LIN {X 0,Y 433.685,Z 905.49,A -85,B 0,C 180,E1 20760.988,E2 20760.988} C_VEL
LIN {X 0,Y 436.129,Z 886.958,A -85,B 0,C 180,E1 20758.951,E2 20758.951} C_VEL
LIN {X 0,Y 438.677,Z 867.119,A -85,B 0,C 180,E1 20757.103,E2 20757.103} C_VEL
LIN {X 0,Y 441.233,Z 846.822,A -85,B 0,C 180,E1 20755.497,E2 20755.497} C_VEL
LIN {X 0,Y 443.681,Z 826.289,A -85,B 0,C 180,E1 20754.137,E2 20754.137} C_VEL
LIN {X 0,Y 445.995,Z 805.048,A -85,B 0,C 180,E1 20752.996,E2 20752.996} C_VEL
LIN {X 0,Y 448.001,Z 783.649,A -85,B 0,C 180,E1 20752.093,E2 20752.093} C_VEL
LIN {X 0,Y 449.731,Z 761.555,A -85,B 0,C 180,E1 20751.394,E2 20751.394} C_VEL
LIN {X 0,Y 450.869,Z 738.561,A -85,B 0,C 180,E1 20750.885,E2 20750.885} C_VEL
LIN {X 0,Y 457.384,Z 507.602,A -85,B 0,C 180,E1 20746.748,E2 20746.748} C_VEL
LIN {X 0,Y 457.893,Z 484.201,A -85,B 0,C 180,E1 20746.312,E2 20746.312} C_VEL
LIN {X 0,Y 453.524,Z 445.974,A -85,B 0,C 180,E1 20745.004,E2 20745.004} C_VEL
LIN {X 0,Y 454.168,Z 438.034,A -85,B 0,C 180,E1 20744.433,E2 20744.433} C_VEL
LIN {X 0,Y 445.913,Z 418.926,A -85,B 0,C 180,E1 20741.897,E2 20741.897} C_VEL
LIN {X 0,Y 436.713,Z 399.875,A -85,B 0,C 180,E1 20739.021,E2 20739.021} C_VEL
LIN {X 0,Y 429.632,Z 386.565,A -85,B 0,C 180,E1 20736.734,E2 20736.734} C_VEL
LIN {X 0,Y 427.405,Z 382.219,A -85,B 0,C 180,E1 20735.957,E2 20735.957} C_VEL
LIN {X 0,Y 425.494,Z 378.909,A -85,B 0,C 180,E1 20735.314,E2 20735.314} C_VEL
LIN {X 0,Y 425.26,Z 377.8,A -85,B 0,C 180,E1 20735.007,E2 20735.007} C_VEL
LIN {X 0,Y 425.249,Z 377.719,A -85,B 0,C 180,E1 20731.149,E2 20731.149} C_VEL
LIN {X 0,Y 425.285,Z 377.761,A -85,B 0,C 180,E1 20727.59,E2 20727.59} C_VEL
LIN {X 0,Y 425.292,Z 377.705,A -85,B 0,C 180,E1 20723.704,E2 20723.704} C_VEL
LIN {X 0,Y 425.275,Z 377.755,A -85,B 0,C 180,E1 20719.932,E2 20719.932} C_VEL
LIN {X 0,Y 425.243,Z 377.76,A -85,B 0,C 180,E1 20716.248,E2 20716.248} C_VEL
LIN {X 0,Y 425.24,Z 377.762,A -85,B 0,C 180,E1 20712.493,E2 20712.493} C_VEL
LIN {X 0,Y 425.256,Z 377.761,A -85,B 0,C 180,E1 20708.79,E2 20708.79} C_VEL
LIN {X 0,Y 425.295,Z 377.761,A -85,B 0,C 180,E1 20705.125,E2 20705.125} C_VEL
LIN {X 0,Y 425.3,Z 377.754,A -85,B 0,C 180,E1 20701.212,E2 20701.212} C_VEL
LIN {X 0,Y 425.271,Z 377.747,A -85,B 0,C 180,E1 20697.439,E2 20697.439} C_VEL
LIN {X 0,Y 425.253,Z 377.742,A -85,B 0,C 180,E1 20693.791,E2 20693.791} C_VEL
LIN {X 0,Y 425.259,Z 377.746,A -85,B 0,C 180,E1 20689.98,E2 20689.98} C_VEL
LIN {X 0,Y 425.285,Z 377.751,A -85,B 0,C 180,E1 20686.263,E2 20686.263} C_VEL
LIN {X 0,Y 425.313,Z 377.754,A -85,B 0,C 180,E1 20682.487,E2 20682.487} C_VEL
LIN {X 0,Y 425.318,Z 377.756,A -85,B 0,C 180,E1 20678.565,E2 20678.565} C_VEL
LIN {X 0,Y 425.291,Z 377.76,A -85,B 0,C 180,E1 20674.815,E2 20674.815} C_VEL
LIN {X 0,Y 425.275,Z 377.761,A -85,B 0,C 180,E1 20671.185,E2 20671.185} C_VEL
LIN {X 0,Y 425.278,Z 377.761,A -85,B 0,C 180,E1 20667.265,E2 20667.265} C_VEL
LIN {X 0,Y 425.293,Z 377.749,A -85,B 0,C 180,E1 20663.501,E2 20663.501} C_VEL
LIN {X 0,Y 425.318,Z 377.722,A -85,B 0,C 180,E1 20659.723,E2 20659.723} C_VEL
LIN {X 0,Y 425.314,Z 377.711,A -85,B 0,C 180,E1 20655.904,E2 20655.904} C_VEL
LIN {X 0,Y 425.346,Z 378.092,A -85,B 0,C 180,E1 20655.176,E2 20655.176} C_VEL
LIN {X 0,Y 426.901,Z 381.643,A -85,B 0,C 180,E1 20654.41,E2 20654.41} C_VEL
LIN {X 0,Y 433.072,Z 394.451,A -85,B 0,C 180,E1 20651.877,E2 20651.877} C_VEL
LIN {X 0,Y 446.756,Z 414.799,A -85,B 0,C 180,E1 20649.706,E2 20649.706} C_VEL
LIN {X 0,Y 455.763,Z 429.646,A -85,B 0,C 180,E1 20648.363,E2 20648.363} C_VEL
LIN {X 0,Y 450.641,Z 657.309,A -85,B 0,C 180,E1 20644.565,E2 20644.565} C_VEL
LIN {X 0,Y 450.433,Z 662.808,A -85,B 0,C 180,E1 20644.428,E2 20644.428} C_VEL
LIN {X 0,Y 449.038,Z 671.512,A -85,B 0,C 180,E1 20644.293,E2 20644.293} C_VEL
LIN {X 0,Y 443.452,Z 689.634,A -85,B 0,C 180,E1 20644.11,E2 20644.11} C_VEL
LIN {X 0,Y 442.087,Z 696.982,A -85,B 0,C 180,E1 20643.867,E2 20643.867} C_VEL
LIN {X 0,Y 440.387,Z 715.115,A -85,B 0,C 180,E1 20642.936,E2 20642.936} C_VEL
LIN {X 0,Y 438.178,Z 733.664,A -85,B 0,C 180,E1 20641.729,E2 20641.729} C_VEL
LIN {X 0,Y 435.687,Z 751.205,A -85,B 0,C 180,E1 20640.319,E2 20640.319} C_VEL
LIN {X 0,Y 433.01,Z 767.859,A -85,B 0,C 180,E1 20638.701,E2 20638.701} C_VEL
LIN {X 0,Y 430.37,Z 783.046,A -85,B 0,C 180,E1 20636.935,E2 20636.935} C_VEL
LIN {X 0,Y 427.782,Z 796.911,A -85,B 0,C 180,E1 20635.024,E2 20635.024} C_VEL
LIN {X 0,Y 425.201,Z 810.306,A -85,B 0,C 180,E1 20632.811,E2 20632.811} C_VEL
LIN {X 0,Y 422.915,Z 822.107,A -85,B 0,C 180,E1 20630.479,E2 20630.479} C_VEL
LIN {X 0,Y 420.863,Z 833.129,A -85,B 0,C 180,E1 20627.844,E2 20627.844} C_VEL
LIN {X 0,Y 419.312,Z 842.132,A -85,B 0,C 180,E1 20625.204,E2 20625.204} C_VEL
LIN {X 0,Y 418.149,Z 849.722,A -85,B 0,C 180,E1 20622.426,E2 20622.426} C_VEL
LIN {X 0,Y 417.374,Z 855.822,A -85,B 0,C 180,E1 20619.513,E2 20619.513} C_VEL
LIN {X 0,Y 416.934,Z 860.132,A -85,B 0,C 180,E1 20616.609,E2 20616.609} C_VEL
LIN {X 0,Y 416.685,Z 862.845,A -85,B 0,C 180,E1 20613.714,E2 20613.714} C_VEL
LIN {X 0,Y 416.609,Z 864.041,A -85,B 0,C 180,E1 20610.825,E2 20610.825} C_VEL
LIN {X 0,Y 416.631,Z 863.76,A -85,B 0,C 180,E1 20607.937,E2 20607.937} C_VEL
LIN {X 0,Y 416.768,Z 861.992,A -85,B 0,C 180,E1 20605.045,E2 20605.045} C_VEL
LIN {X 0,Y 417.074,Z 858.614,A -85,B 0,C 180,E1 20602.146,E2 20602.146} C_VEL
LIN {X 0,Y 417.623,Z 853.58,A -85,B 0,C 180,E1 20599.238,E2 20599.238} C_VEL
LIN {X 0,Y 418.526,Z 847.119,A -85,B 0,C 180,E1 20596.461,E2 20596.461} C_VEL
LIN {X 0,Y 419.849,Z 838.866,A -85,B 0,C 180,E1 20593.68,E2 20593.68} C_VEL
LIN {X 0,Y 421.61,Z 829.134,A -85,B 0,C 180,E1 20591.042,E2 20591.042} C_VEL
LIN {X 0,Y 423.73,Z 817.946,A -85,B 0,C 180,E1 20588.548,E2 20588.548} C_VEL
LIN {X 0,Y 426.239,Z 805.107,A -85,B 0,C 180,E1 20586.185,E2 20586.185} C_VEL
LIN {X 0,Y 428.744,Z 791.813,A -85,B 0,C 180,E1 20584.147,E2 20584.147} C_VEL
LIN {X 0,Y 431.518,Z 776.647,A -85,B 0,C 180,E1 20582.192,E2 20582.192} C_VEL
LIN {X 0,Y 434.306,Z 760.066,A -85,B 0,C 180,E1 20580.411,E2 20580.411} C_VEL
LIN {X 0,Y 436.848,Z 743.483,A -85,B 0,C 180,E1 20578.93,E2 20578.93} C_VEL
LIN {X 0,Y 439.262,Z 725.247,A -85,B 0,C 180,E1 20577.596,E2 20577.596} C_VEL
LIN {X 0,Y 441.256,Z 706.44,A -85,B 0,C 180,E1 20576.498,E2 20576.498} C_VEL
LIN {X 0,Y 442.866,Z 686.886,A -85,B 0,C 180,E1 20575.612,E2 20575.612} C_VEL
LIN {X 0,Y 444.042,Z 666.143,A -85,B 0,C 180,E1 20574.926,E2 20574.926} C_VEL
LIN {X 0,Y 444.645,Z 645.299,A -85,B 0,C 180,E1 20574.471,E2 20574.471} C_VEL
LIN {X 0,Y 449.744,Z 432.69,A -85,B 0,C 180,E1 20570.911,E2 20570.911} C_VEL
LIN {X 0,Y 437.485,Z 413.17,A -85,B 0,C 180,E1 20569.011,E2 20569.011} C_VEL
LIN {X 0,Y 425.475,Z 395.725,A -85,B 0,C 180,E1 20567.007,E2 20567.007} C_VEL
LIN {X 0,Y 423.728,Z 392.497,A -85,B 0,C 180,E1 20566.421,E2 20566.421} C_VEL
LIN {X 0,Y 420.654,Z 386.269,A -85,B 0,C 180,E1 20565.099,E2 20565.099} C_VEL
LIN {X 0,Y 418.847,Z 382.419,A -85,B 0,C 180,E1 20564.268,E2 20564.268} C_VEL
LIN {X 0,Y 417.377,Z 378.887,A -85,B 0,C 180,E1 20563.435,E2 20563.435} C_VEL
LIN {X 0,Y 417.361,Z 378.7,A -85,B 0,C 180,E1 20559.587,E2 20559.587} C_VEL
LIN {X 0,Y 417.377,Z 378.748,A -85,B 0,C 180,E1 20555.706,E2 20555.706} C_VEL
LIN {X 0,Y 417.384,Z 378.739,A -85,B 0,C 180,E1 20551.752,E2 20551.752} C_VEL
LIN {X 0,Y 417.384,Z 378.735,A -85,B 0,C 180,E1 20547.848,E2 20547.848} C_VEL
LIN {X 0,Y 417.354,Z 378.738,A -85,B 0,C 180,E1 20544.034,E2 20544.034} C_VEL
LIN {X 0,Y 417.335,Z 378.745,A -85,B 0,C 180,E1 20540.328,E2 20540.328} C_VEL
LIN {X 0,Y 417.33,Z 378.747,A -85,B 0,C 180,E1 20536.422,E2 20536.422} C_VEL
LIN {X 0,Y 417.334,Z 378.75,A -85,B 0,C 180,E1 20532.593,E2 20532.593} C_VEL
LIN {X 0,Y 417.352,Z 378.746,A -85,B 0,C 180,E1 20528.82,E2 20528.82} C_VEL
LIN {X 0,Y 417.366,Z 378.732,A -85,B 0,C 180,E1 20525.086,E2 20525.086} C_VEL
LIN {X 0,Y 417.348,Z 378.73,A -85,B 0,C 180,E1 20521.236,E2 20521.236} C_VEL
LIN {X 0,Y 417.317,Z 378.736,A -85,B 0,C 180,E1 20517.529,E2 20517.529} C_VEL
LIN {X 0,Y 417.309,Z 378.744,A -85,B 0,C 180,E1 20513.811,E2 20513.811} C_VEL
LIN {X 0,Y 417.318,Z 378.747,A -85,B 0,C 180,E1 20510.067,E2 20510.067} C_VEL
LIN {X 0,Y 417.34,Z 378.747,A -85,B 0,C 180,E1 20506.28,E2 20506.28} C_VEL
LIN {X 0,Y 417.35,Z 378.746,A -85,B 0,C 180,E1 20502.431,E2 20502.431} C_VEL
LIN {X 0,Y 417.344,Z 378.742,A -85,B 0,C 180,E1 20498.497,E2 20498.497} C_VEL
LIN {X 0,Y 417.314,Z 378.704,A -85,B 0,C 180,E1 20494.756,E2 20494.756} C_VEL
LIN {X 0,Y 417.305,Z 378.719,A -85,B 0,C 180,E1 20491.054,E2 20491.054} C_VEL
LIN {X 0,Y 417.315,Z 378.746,A -85,B 0,C 180,E1 20487.216,E2 20487.216} C_VEL
LIN {X 0,Y 417.397,Z 379.019,A -85,B 0,C 180,E1 20486.114,E2 20486.114} C_VEL
LIN {X 0,Y 418.946,Z 382.633,A -85,B 0,C 180,E1 20485.389,E2 20485.389} C_VEL
LIN {X 0,Y 420.122,Z 384.448,A -85,B 0,C 180,E1 20485.001,E2 20485.001} C_VEL
LIN {X 0,Y 423.049,Z 390.051,A -85,B 0,C 180,E1 20483.95,E2 20483.95} C_VEL
LIN {X 0,Y 429.251,Z 401.502,A -85,B 0,C 180,E1 20481.884,E2 20481.884} C_VEL
LIN {X 0,Y 438.343,Z 420.229,A -85,B 0,C 180,E1 20478.934,E2 20478.934} C_VEL
LIN {X 0,Y 446.423,Z 438.688,A -85,B 0,C 180,E1 20476.384,E2 20476.384} C_VEL
LIN {X 0,Y 447.647,Z 441.768,A -85,B 0,C 180,E1 20475.984,E2 20475.984} C_VEL
LIN {X 0,Y 447.363,Z 446.602,A -85,B 0,C 180,E1 20475.669,E2 20475.669} C_VEL
LIN {X 0,Y 451.886,Z 487.98,A -85,B 0,C 180,E1 20474.26,E2 20474.26} C_VEL
LIN {X 0,Y 445.169,Z 710.903,A -85,B 0,C 180,E1 20470.217,E2 20470.217} C_VEL
LIN {X 0,Y 443.781,Z 752.109,A -85,B 0,C 180,E1 20469.431,E2 20469.431} C_VEL
LIN {X 0,Y 442.112,Z 774.52,A -85,B 0,C 180,E1 20468.802,E2 20468.802} C_VEL
LIN {X 0,Y 440.035,Z 796.219,A -85,B 0,C 180,E1 20467.959,E2 20467.959} C_VEL
LIN {X 0,Y 437.636,Z 818.272,A -85,B 0,C 180,E1 20466.847,E2 20466.847} C_VEL
LIN {X 0,Y 435.085,Z 839.09,A -85,B 0,C 180,E1 20465.546,E2 20465.546} C_VEL
LIN {X 0,Y 432.405,Z 859.055,A -85,B 0,C 180,E1 20464.023,E2 20464.023} C_VEL
LIN {X 0,Y 429.758,Z 878.3,A -85,B 0,C 180,E1 20462.285,E2 20462.285} C_VEL
LIN {X 0,Y 427.222,Z 896.559,A -85,B 0,C 180,E1 20460.363,E2 20460.363} C_VEL
LIN {X 0,Y 424.728,Z 914.512,A -85,B 0,C 180,E1 20458.162,E2 20458.162} C_VEL
LIN {X 0,Y 422.653,Z 929.899,A -85,B 0,C 180,E1 20455.952,E2 20455.952} C_VEL
LIN {X 0,Y 420.762,Z 944.814,A -85,B 0,C 180,E1 20453.473,E2 20453.473} C_VEL
LIN {X 0,Y 419.245,Z 957.761,A -85,B 0,C 180,E1 20450.959,E2 20450.959} C_VEL
LIN {X 0,Y 418.024,Z 969.386,A -85,B 0,C 180,E1 20448.275,E2 20448.275} C_VEL
LIN {X 0,Y 417.121,Z 979.673,A -85,B 0,C 180,E1 20445.43,E2 20445.43} C_VEL
LIN {X 0,Y 416.535,Z 988.002,A -85,B 0,C 180,E1 20442.616,E2 20442.616} C_VEL
LIN {X 0,Y 416.213,Z 994.134,A -85,B 0,C 180,E1 20439.96,E2 20439.96} C_VEL
LIN {X 0,Y 416.05,Z 999.088,A -85,B 0,C 180,E1 20437.179,E2 20437.179} C_VEL
LIN {X 0,Y 416.009,Z 1002.29,A -85,B 0,C 180,E1 20434.411,E2 20434.411} C_VEL
LIN {X 0,Y 415.985,Z 1004.039,A -85,B 0,C 180,E1 20431.653,E2 20431.653} C_VEL
LIN {X 0,Y 415.985,Z 1004.171,A -85,B 0,C 180,E1 20429.037,E2 20429.037} C_VEL
LIN {X 0,Y 415.999,Z 1002.917,A -85,B 0,C 180,E1 20426.28,E2 20426.28} C_VEL
LIN {X 0,Y 416.049,Z 999.992,A -85,B 0,C 180,E1 20423.516,E2 20423.516} C_VEL
LIN {X 0,Y 416.17,Z 995.273,A -85,B 0,C 180,E1 20420.599,E2 20420.599} C_VEL
LIN {X 0,Y 416.466,Z 989.401,A -85,B 0,C 180,E1 20417.946,E2 20417.946} C_VEL
LIN {X 0,Y 416.975,Z 981.346,A -85,B 0,C 180,E1 20415.093,E2 20415.093} C_VEL
LIN {X 0,Y 417.747,Z 972.262,A -85,B 0,C 180,E1 20412.45,E2 20412.45} C_VEL
LIN {X 0,Y 418.881,Z 961.013,A -85,B 0,C 180,E1 20409.753,E2 20409.753} C_VEL
LIN {X 0,Y 420.406,Z 947.649,A -85,B 0,C 180,E1 20407.046,E2 20407.046} C_VEL
LIN {X 0,Y 422.175,Z 933.639,A -85,B 0,C 180,E1 20404.62,E2 20404.62} C_VEL
LIN {X 0,Y 424.314,Z 917.663,A -85,B 0,C 180,E1 20402.268,E2 20402.268} C_VEL
LIN {X 0,Y 426.706,Z 900.197,A -85,B 0,C 180,E1 20400.063,E2 20400.063} C_VEL
LIN {X 0,Y 429.342,Z 881.231,A -85,B 0,C 180,E1 20398.002,E2 20398.002} C_VEL
LIN {X 0,Y 431.97,Z 862.482,A -85,B 0,C 180,E1 20396.258,E2 20396.258} C_VEL
LIN {X 0,Y 434.568,Z 842.892,A -85,B 0,C 180,E1 20394.73,E2 20394.73} C_VEL
LIN {X 0,Y 437.204,Z 821.8,A -85,B 0,C 180,E1 20393.357,E2 20393.357} C_VEL
LIN {X 0,Y 439.618,Z 800.623,A -85,B 0,C 180,E1 20392.239,E2 20392.239} C_VEL
LIN {X 0,Y 441.709,Z 778.929,A -85,B 0,C 180,E1 20391.349,E2 20391.349} C_VEL
LIN {X 0,Y 443.471,Z 756.618,A -85,B 0,C 180,E1 20390.683,E2 20390.683} C_VEL
LIN {X 0,Y 444.644,Z 728.865,A -85,B 0,C 180,E1 20390.109,E2 20390.109} C_VEL
LIN {X 0,Y 451.52,Z 499.275,A -85,B 0,C 180,E1 20385.945,E2 20385.945} C_VEL
LIN {X 0,Y 451.746,Z 485.372,A -85,B 0,C 180,E1 20385.672,E2 20385.672} C_VEL
LIN {X 0,Y 447.267,Z 445.505,A -85,B 0,C 180,E1 20384.288,E2 20384.288} C_VEL
LIN {X 0,Y 447.594,Z 441.595,A -85,B 0,C 180,E1 20384.005,E2 20384.005} C_VEL
LIN {X 0,Y 439.941,Z 423.676,A -85,B 0,C 180,E1 20381.577,E2 20381.577} C_VEL
LIN {X 0,Y 431.185,Z 405.327,A -85,B 0,C 180,E1 20378.762,E2 20378.762} C_VEL
LIN {X 0,Y 424.17,Z 392.045,A -85,B 0,C 180,E1 20376.442,E2 20376.442} C_VEL
LIN {X 0,Y 421.752,Z 387.543,A -85,B 0,C 180,E1 20375.603,E2 20375.603} C_VEL
LIN {X 0,Y 419.323,Z 383.098,A -85,B 0,C 180,E1 20374.742,E2 20374.742} C_VEL
LIN {X 0,Y 417.552,Z 379.73,A -85,B 0,C 180,E1 20374.078,E2 20374.078} C_VEL
LIN {X 0,Y 417.352,Z 378.764,A -85,B 0,C 180,E1 20373.766,E2 20373.766} C_VEL
LIN {X 0,Y 417.365,Z 378.696,A -85,B 0,C 180,E1 20369.873,E2 20369.873} C_VEL
LIN {X 0,Y 417.334,Z 378.721,A -85,B 0,C 180,E1 20366.157,E2 20366.157} C_VEL
LIN {X 0,Y 417.309,Z 378.722,A -85,B 0,C 180,E1 20362.371,E2 20362.371} C_VEL
LIN {X 0,Y 417.3,Z 378.741,A -85,B 0,C 180,E1 20358.582,E2 20358.582} C_VEL
LIN {X 0,Y 417.3,Z 378.742,A -85,B 0,C 180,E1 20354.713,E2 20354.713} C_VEL
LIN {X 0,Y 417.328,Z 378.735,A -85,B 0,C 180,E1 20351.05,E2 20351.05} C_VEL
LIN {X 0,Y 417.366,Z 378.73,A -85,B 0,C 180,E1 20347.294,E2 20347.294} C_VEL
LIN {X 0,Y 417.341,Z 378.735,A -85,B 0,C 180,E1 20343.433,E2 20343.433} C_VEL
LIN {X 0,Y 417.32,Z 378.748,A -85,B 0,C 180,E1 20339.725,E2 20339.725} C_VEL
LIN {X 0,Y 417.316,Z 378.75,A -85,B 0,C 180,E1 20335.878,E2 20335.878} C_VEL
LIN {X 0,Y 417.319,Z 378.748,A -85,B 0,C 180,E1 20332.012,E2 20332.012} C_VEL
LIN {X 0,Y 417.338,Z 378.742,A -85,B 0,C 180,E1 20328.25,E2 20328.25} C_VEL
LIN {X 0,Y 417.367,Z 378.733,A -85,B 0,C 180,E1 20324.436,E2 20324.436} C_VEL
LIN {X 0,Y 417.374,Z 378.73,A -85,B 0,C 180,E1 20320.549,E2 20320.549} C_VEL
LIN {X 0,Y 417.36,Z 378.732,A -85,B 0,C 180,E1 20316.716,E2 20316.716} C_VEL
LIN {X 0,Y 417.342,Z 378.734,A -85,B 0,C 180,E1 20312.922,E2 20312.922} C_VEL
LIN {X 0,Y 417.336,Z 378.735,A -85,B 0,C 180,E1 20309.156,E2 20309.156} C_VEL
LIN {X 0,Y 417.341,Z 378.741,A -85,B 0,C 180,E1 20305.236,E2 20305.236} C_VEL
LIN {X 0,Y 417.354,Z 378.695,A -85,B 0,C 180,E1 20301.473,E2 20301.473} C_VEL
LIN {X 0,Y 417.376,Z 378.728,A -85,B 0,C 180,E1 20297.688,E2 20297.688} C_VEL
LIN {X 0,Y 417.386,Z 378.957,A -85,B 0,C 180,E1 20296.428,E2 20296.428} C_VEL
LIN {X 0,Y 418.856,Z 382.432,A -85,B 0,C 180,E1 20295.619,E2 20295.619} C_VEL
LIN {X 0,Y 423.562,Z 392.072,A -85,B 0,C 180,E1 20293.555,E2 20293.555} C_VEL
LIN {X 0,Y 425.441,Z 395.688,A -85,B 0,C 180,E1 20292.889,E2 20292.889} C_VEL
LIN {X 0,Y 438.264,Z 414.369,A -85,B 0,C 180,E1 20290.762,E2 20290.762} C_VEL
LIN {X 0,Y 449.714,Z 432.708,A -85,B 0,C 180,E1 20288.991,E2 20288.991} C_VEL
LIN {X 0,Y 444.324,Z 658.235,A -85,B 0,C 180,E1 20285.184,E2 20285.184} C_VEL
LIN {X 0,Y 443.397,Z 678.464,A -85,B 0,C 180,E1 20284.606,E2 20284.606} C_VEL
LIN {X 0,Y 442.087,Z 696.982,A -85,B 0,C 180,E1 20283.867,E2 20283.867} C_VEL
LIN {X 0,Y 440.669,Z 704.442,A -85,B 0,C 180,E1 20283.597,E2 20283.597} C_VEL
LIN {X 0,Y 433.955,Z 722.866,A -85,B 0,C 180,E1 20283.048,E2 20283.048} C_VEL
LIN {X 0,Y 432.274,Z 729.797,A -85,B 0,C 180,E1 20282.669,E2 20282.669} C_VEL
LIN {X 0,Y 429.796,Z 747.41,A -85,B 0,C 180,E1 20281.324,E2 20281.324} C_VEL
LIN {X 0,Y 427.07,Z 764.295,A -85,B 0,C 180,E1 20279.754,E2 20279.754} C_VEL
LIN {X 0,Y 424.194,Z 780.169,A -85,B 0,C 180,E1 20277.97,E2 20277.97} C_VEL
LIN {X 0,Y 421.39,Z 794.612,A -85,B 0,C 180,E1 20276.034,E2 20276.034} C_VEL
LIN {X 0,Y 418.587,Z 808.542,A -85,B 0,C 180,E1 20273.805,E2 20273.805} C_VEL
LIN {X 0,Y 416.181,Z 820.323,A -85,B 0,C 180,E1 20271.563,E2 20271.563} C_VEL
LIN {X 0,Y 413.975,Z 831.353,A -85,B 0,C 180,E1 20269.027,E2 20269.027} C_VEL
LIN {X 0,Y 412.129,Z 840.904,A -85,B 0,C 180,E1 20266.343,E2 20266.343} C_VEL
LIN {X 0,Y 410.801,Z 848.632,A -85,B 0,C 180,E1 20263.654,E2 20263.654} C_VEL
LIN {X 0,Y 409.786,Z 855.313,A -85,B 0,C 180,E1 20260.685,E2 20260.685} C_VEL
LIN {X 0,Y 409.23,Z 860.026,A -85,B 0,C 180,E1 20257.863,E2 20257.863} C_VEL
LIN {X 0,Y 408.896,Z 863.375,A -85,B 0,C 180,E1 20254.909,E2 20254.909} C_VEL
LIN {X 0,Y 408.744,Z 865.11,A -85,B 0,C 180,E1 20251.962,E2 20251.962} C_VEL
LIN {X 0,Y 408.721,Z 865.363,A -85,B 0,C 180,E1 20249.018,E2 20249.018} C_VEL
LIN {X 0,Y 408.82,Z 864.049,A -85,B 0,C 180,E1 20245.933,E2 20245.933} C_VEL
LIN {X 0,Y 409.104,Z 861.239,A -85,B 0,C 180,E1 20242.981,E2 20242.981} C_VEL
LIN {X 0,Y 409.6,Z 856.837,A -85,B 0,C 180,E1 20240.02,E2 20240.02} C_VEL
LIN {X 0,Y 410.491,Z 850.674,A -85,B 0,C 180,E1 20237.051,E2 20237.051} C_VEL
LIN {X 0,Y 411.77,Z 842.969,A -85,B 0,C 180,E1 20234.22,E2 20234.22} C_VEL
LIN {X 0,Y 413.475,Z 833.831,A -85,B 0,C 180,E1 20231.533,E2 20231.533} C_VEL
LIN {X 0,Y 415.565,Z 823.305,A -85,B 0,C 180,E1 20228.994,E2 20228.994} C_VEL
LIN {X 0,Y 418.019,Z 811.385,A -85,B 0,C 180,E1 20226.608,E2 20226.608} C_VEL
LIN {X 0,Y 420.734,Z 798.043,A -85,B 0,C 180,E1 20224.375,E2 20224.375} C_VEL
LIN {X 0,Y 423.676,Z 783.109,A -85,B 0,C 180,E1 20222.298,E2 20222.298} C_VEL
LIN {X 0,Y 426.477,Z 767.657,A -85,B 0,C 180,E1 20220.508,E2 20220.508} C_VEL
LIN {X 0,Y 429.291,Z 750.669,A -85,B 0,C 180,E1 20218.868,E2 20218.868} C_VEL
LIN {X 0,Y 431.966,Z 732.255,A -85,B 0,C 180,E1 20217.41,E2 20217.41} C_VEL
LIN {X 0,Y 434.217,Z 713.799,A -85,B 0,C 180,E1 20216.229,E2 20216.229} C_VEL
LIN {X 0,Y 436.039,Z 694.688,A -85,B 0,C 180,E1 20215.266,E2 20215.266} C_VEL
LIN {X 0,Y 437.385,Z 674.644,A -85,B 0,C 180,E1 20214.513,E2 20214.513} C_VEL
LIN {X 0,Y 438.203,Z 654.336,A -85,B 0,C 180,E1 20213.988,E2 20213.988} C_VEL
LIN {X 0,Y 443.705,Z 435.902,A -85,B 0,C 180,E1 20210.263,E2 20210.263} C_VEL
LIN {X 0,Y 432.287,Z 417.811,A -85,B 0,C 180,E1 20208.439,E2 20208.439} C_VEL
LIN {X 0,Y 420.875,Z 401.15,A -85,B 0,C 180,E1 20206.484,E2 20206.484} C_VEL
LIN {X 0,Y 417.002,Z 395.788,A -85,B 0,C 180,E1 20205.759,E2 20205.759} C_VEL
LIN {X 0,Y 413.044,Z 387.675,A -85,B 0,C 180,E1 20204.007,E2 20204.007} C_VEL
LIN {X 0,Y 411.129,Z 383.746,A -85,B 0,C 180,E1 20203.109,E2 20203.109} C_VEL
LIN {X 0,Y 409.528,Z 380.273,A -85,B 0,C 180,E1 20202.294,E2 20202.294} C_VEL
LIN {X 0,Y 409.441,Z 379.726,A -85,B 0,C 180,E1 20201.863,E2 20201.863} C_VEL
LIN {X 0,Y 409.439,Z 379.683,A -85,B 0,C 180,E1 20197.936,E2 20197.936} C_VEL
LIN {X 0,Y 409.44,Z 379.721,A -85,B 0,C 180,E1 20194.002,E2 20194.002} C_VEL
LIN {X 0,Y 409.425,Z 379.721,A -85,B 0,C 180,E1 20190.183,E2 20190.183} C_VEL
LIN {X 0,Y 409.404,Z 379.724,A -85,B 0,C 180,E1 20186.391,E2 20186.391} C_VEL
LIN {X 0,Y 409.395,Z 379.724,A -85,B 0,C 180,E1 20182.547,E2 20182.547} C_VEL
LIN {X 0,Y 409.395,Z 379.723,A -85,B 0,C 180,E1 20178.645,E2 20178.645} C_VEL
LIN {X 0,Y 409.407,Z 379.72,A -85,B 0,C 180,E1 20174.859,E2 20174.859} C_VEL
LIN {X 0,Y 409.429,Z 379.719,A -85,B 0,C 180,E1 20171.124,E2 20171.124} C_VEL
LIN {X 0,Y 409.44,Z 379.722,A -85,B 0,C 180,E1 20167.155,E2 20167.155} C_VEL
LIN {X 0,Y 409.415,Z 379.733,A -85,B 0,C 180,E1 20163.22,E2 20163.22} C_VEL
LIN {X 0,Y 409.391,Z 379.739,A -85,B 0,C 180,E1 20159.441,E2 20159.441} C_VEL
LIN {X 0,Y 409.374,Z 379.739,A -85,B 0,C 180,E1 20155.658,E2 20155.658} C_VEL
LIN {X 0,Y 409.369,Z 379.736,A -85,B 0,C 180,E1 20151.715,E2 20151.715} C_VEL
LIN {X 0,Y 409.371,Z 379.732,A -85,B 0,C 180,E1 20147.875,E2 20147.875} C_VEL
LIN {X 0,Y 409.389,Z 379.728,A -85,B 0,C 180,E1 20144.125,E2 20144.125} C_VEL
LIN {X 0,Y 409.41,Z 379.727,A -85,B 0,C 180,E1 20140.305,E2 20140.305} C_VEL
LIN {X 0,Y 409.391,Z 379.684,A -85,B 0,C 180,E1 20136.541,E2 20136.541} C_VEL
LIN {X 0,Y 409.38,Z 379.744,A -85,B 0,C 180,E1 20132.741,E2 20132.741} C_VEL
LIN {X 0,Y 409.367,Z 379.692,A -85,B 0,C 180,E1 20128.979,E2 20128.979} C_VEL
LIN {X 0,Y 409.408,Z 379.868,A -85,B 0,C 180,E1 20127.501,E2 20127.501} C_VEL
LIN {X 0,Y 409.655,Z 381.055,A -85,B 0,C 180,E1 20127.191,E2 20127.191} C_VEL
LIN {X 0,Y 411.437,Z 384.158,A -85,B 0,C 180,E1 20126.52,E2 20126.52} C_VEL
LIN {X 0,Y 412.223,Z 385.277,A -85,B 0,C 180,E1 20126.259,E2 20126.259} C_VEL
LIN {X 0,Y 414.379,Z 389.245,A -85,B 0,C 180,E1 20125.457,E2 20125.457} C_VEL
LIN {X 0,Y 421.912,Z 403.539,A -85,B 0,C 180,E1 20122.768,E2 20122.768} C_VEL
LIN {X 0,Y 429.754,Z 419.216,A -85,B 0,C 180,E1 20120.148,E2 20120.148} C_VEL
LIN {X 0,Y 437.914,Z 437.424,A -85,B 0,C 180,E1 20117.481,E2 20117.481} C_VEL
LIN {X 0,Y 441.155,Z 445.468,A -85,B 0,C 180,E1 20116.438,E2 20116.438} C_VEL
LIN {X 0,Y 445.818,Z 489.253,A -85,B 0,C 180,E1 20114.913,E2 20114.913} C_VEL
LIN {X 0,Y 438.748,Z 711.806,A -85,B 0,C 180,E1 20110.827,E2 20110.827} C_VEL
LIN {X 0,Y 437.332,Z 751.282,A -85,B 0,C 180,E1 20110.061,E2 20110.061} C_VEL
LIN {X 0,Y 435.603,Z 773.536,A -85,B 0,C 180,E1 20109.429,E2 20109.429} C_VEL
LIN {X 0,Y 433.377,Z 795.43,A -85,B 0,C 180,E1 20108.568,E2 20108.568} C_VEL
LIN {X 0,Y 430.842,Z 817.417,A -85,B 0,C 180,E1 20107.443,E2 20107.443} C_VEL
LIN {X 0,Y 428.301,Z 837.149,A -85,B 0,C 180,E1 20106.197,E2 20106.197} C_VEL
LIN {X 0,Y 425.429,Z 857.197,A -85,B 0,C 180,E1 20104.656,E2 20104.656} C_VEL
LIN {X 0,Y 422.501,Z 877.307,A -85,B 0,C 180,E1 20102.812,E2 20102.812} C_VEL
LIN {X 0,Y 419.725,Z 895.905,A -85,B 0,C 180,E1 20100.805,E2 20100.805} C_VEL
LIN {X 0,Y 417.133,Z 913.427,A -85,B 0,C 180,E1 20098.596,E2 20098.596} C_VEL
LIN {X 0,Y 414.8,Z 929.853,A -85,B 0,C 180,E1 20096.173,E2 20096.173} C_VEL
LIN {X 0,Y 412.885,Z 944.28,A -85,B 0,C 180,E1 20093.701,E2 20093.701} C_VEL
LIN {X 0,Y 411.293,Z 957.4,A -85,B 0,C 180,E1 20091.086,E2 20091.086} C_VEL
LIN {X 0,Y 410.044,Z 968.966,A -85,B 0,C 180,E1 20088.333,E2 20088.333} C_VEL
LIN {X 0,Y 409.144,Z 979.073,A -85,B 0,C 180,E1 20085.447,E2 20085.447} C_VEL
LIN {X 0,Y 408.571,Z 987.276,A -85,B 0,C 180,E1 20082.579,E2 20082.579} C_VEL
LIN {X 0,Y 408.267,Z 993.301,A -85,B 0,C 180,E1 20079.871,E2 20079.871} C_VEL
LIN {X 0,Y 408.144,Z 998.268,A -85,B 0,C 180,E1 20076.894,E2 20076.894} C_VEL
LIN {X 0,Y 408.106,Z 1001.199,A -85,B 0,C 180,E1 20074.215,E2 20074.215} C_VEL
LIN {X 0,Y 408.101,Z 1002.791,A -85,B 0,C 180,E1 20071.264,E2 20071.264} C_VEL
LIN {X 0,Y 408.101,Z 1002.791,A -85,B 0,C 180,E1 20068.737,E2 20068.737} C_VEL
LIN {X 0,Y 408.105,Z 1001.2,A -85,B 0,C 180,E1 20065.786,E2 20065.786} C_VEL
LIN {X 0,Y 408.142,Z 998.268,A -85,B 0,C 180,E1 20063.107,E2 20063.107} C_VEL
LIN {X 0,Y 408.253,Z 993.591,A -85,B 0,C 180,E1 20060.272,E2 20060.272} C_VEL
LIN {X 0,Y 408.553,Z 987.622,A -85,B 0,C 180,E1 20057.565,E2 20057.565} C_VEL
LIN {X 0,Y 409.107,Z 979.53,A -85,B 0,C 180,E1 20054.697,E2 20054.697} C_VEL
LIN {X 0,Y 409.932,Z 970.121,A -85,B 0,C 180,E1 20051.957,E2 20051.957} C_VEL
LIN {X 0,Y 411.139,Z 958.693,A -85,B 0,C 180,E1 20049.206,E2 20049.206} C_VEL
LIN {X 0,Y 412.679,Z 945.861,A -85,B 0,C 180,E1 20046.591,E2 20046.591} C_VEL
LIN {X 0,Y 414.555,Z 931.67,A -85,B 0,C 180,E1 20044.109,E2 20044.109} C_VEL
LIN {X 0,Y 416.947,Z 914.697,A -85,B 0,C 180,E1 20041.578,E2 20041.578} C_VEL
LIN {X 0,Y 419.549,Z 897.118,A -85,B 0,C 180,E1 20039.34,E2 20039.34} C_VEL
LIN {X 0,Y 422.366,Z 878.204,A -85,B 0,C 180,E1 20037.277,E2 20037.277} C_VEL
LIN {X 0,Y 425.2,Z 858.886,A -85,B 0,C 180,E1 20035.483,E2 20035.483} C_VEL
LIN {X 0,Y 428.061,Z 838.761,A -85,B 0,C 180,E1 20033.918,E2 20033.918} C_VEL
LIN {X 0,Y 430.689,Z 818.584,A -85,B 0,C 180,E1 20032.626,E2 20032.626} C_VEL
LIN {X 0,Y 433.288,Z 796.243,A -85,B 0,C 180,E1 20031.469,E2 20031.469} C_VEL
LIN {X 0,Y 435.524,Z 774.394,A -85,B 0,C 180,E1 20030.599,E2 20030.599} C_VEL
LIN {X 0,Y 437.267,Z 752.114,A -85,B 0,C 180,E1 20029.962,E2 20029.962} C_VEL
LIN {X 0,Y 438.573,Z 717.201,A -85,B 0,C 180,E1 20029.274,E2 20029.274} C_VEL
LIN {X 0,Y 445.688,Z 492.711,A -85,B 0,C 180,E1 20025.153,E2 20025.153} C_VEL
LIN {X 0,Y 445.643,Z 486.41,A -85,B 0,C 180,E1 20025.01,E2 20025.01} C_VEL
LIN {X 0,Y 441.098,Z 445.196,A -85,B 0,C 180,E1 20023.558,E2 20023.558} C_VEL
LIN {X 0,Y 433.494,Z 427.387,A -85,B 0,C 180,E1 20021.098,E2 20021.098} C_VEL
LIN {X 0,Y 425.652,Z 410.769,A -85,B 0,C 180,E1 20018.497,E2 20018.497} C_VEL
LIN {X 0,Y 418.321,Z 396.851,A -85,B 0,C 180,E1 20016.013,E2 20016.013} C_VEL
LIN {X 0,Y 414.317,Z 389.182,A -85,B 0,C 180,E1 20014.549,E2 20014.549} C_VEL
LIN {X 0,Y 412.176,Z 385.171,A -85,B 0,C 180,E1 20013.745,E2 20013.745} C_VEL
LIN {X 0,Y 409.893,Z 381.741,A -85,B 0,C 180,E1 20012.954,E2 20012.954} C_VEL
LIN {X 0,Y 409.427,Z 380.028,A -85,B 0,C 180,E1 20012.603,E2 20012.603} C_VEL
LIN {X 0,Y 409.372,Z 379.688,A -85,B 0,C 180,E1 20010.694,E2 20010.694} C_VEL
LIN {X 0,Y 409.37,Z 379.734,A -85,B 0,C 180,E1 20006.862,E2 20006.862} C_VEL
LIN {X 0,Y 409.367,Z 379.694,A -85,B 0,C 180,E1 20002.971,E2 20002.971} C_VEL
LIN {X 0,Y 409.387,Z 379.726,A -85,B 0,C 180,E1 19999.251,E2 19999.251} C_VEL
LIN {X 0,Y 409.413,Z 379.722,A -85,B 0,C 180,E1 19995.438,E2 19995.438} C_VEL
LIN {X 0,Y 409.404,Z 379.722,A -85,B 0,C 180,E1 19991.552,E2 19991.552} C_VEL
LIN {X 0,Y 409.384,Z 379.726,A -85,B 0,C 180,E1 19987.719,E2 19987.719} C_VEL
LIN {X 0,Y 409.374,Z 379.734,A -85,B 0,C 180,E1 19983.921,E2 19983.921} C_VEL
LIN {X 0,Y 409.373,Z 379.741,A -85,B 0,C 180,E1 19980.14,E2 19980.14} C_VEL
LIN {X 0,Y 409.386,Z 379.739,A -85,B 0,C 180,E1 19976.359,E2 19976.359} C_VEL
LIN {X 0,Y 409.412,Z 379.728,A -85,B 0,C 180,E1 19972.563,E2 19972.563} C_VEL
LIN {X 0,Y 409.427,Z 379.719,A -85,B 0,C 180,E1 19968.733,E2 19968.733} C_VEL
LIN {X 0,Y 409.423,Z 379.718,A -85,B 0,C 180,E1 19964.852,E2 19964.852} C_VEL
LIN {X 0,Y 409.403,Z 379.722,A -85,B 0,C 180,E1 19961.045,E2 19961.045} C_VEL
LIN {X 0,Y 409.392,Z 379.725,A -85,B 0,C 180,E1 19957.301,E2 19957.301} C_VEL
LIN {X 0,Y 409.395,Z 379.725,A -85,B 0,C 180,E1 19953.352,E2 19953.352} C_VEL
LIN {X 0,Y 409.403,Z 379.723,A -85,B 0,C 180,E1 19949.543,E2 19949.543} C_VEL
LIN {X 0,Y 409.429,Z 379.722,A -85,B 0,C 180,E1 19945.828,E2 19945.828} C_VEL
LIN {X 0,Y 409.439,Z 379.683,A -85,B 0,C 180,E1 19942.019,E2 19942.019} C_VEL
LIN {X 0,Y 409.437,Z 379.73,A -85,B 0,C 180,E1 19938.136,E2 19938.136} C_VEL
LIN {X 0,Y 409.497,Z 380.129,A -85,B 0,C 180,E1 19937.631,E2 19937.631} C_VEL
LIN {X 0,Y 410.901,Z 383.458,A -85,B 0,C 180,E1 19936.861,E2 19936.861} C_VEL
LIN {X 0,Y 411.907,Z 385.288,A -85,B 0,C 180,E1 19936.419,E2 19936.419} C_VEL
LIN {X 0,Y 416.601,Z 395.006,A -85,B 0,C 180,E1 19934.293,E2 19934.293} C_VEL
LIN {X 0,Y 418.312,Z 397.656,A -85,B 0,C 180,E1 19933.871,E2 19933.871} C_VEL
LIN {X 0,Y 428.876,Z 412.733,A -85,B 0,C 180,E1 19932.027,E2 19932.027} C_VEL
LIN {X 0,Y 440.53,Z 430.73,A -85,B 0,C 180,E1 19930.129,E2 19930.129} C_VEL
LIN {X 0,Y 443.724,Z 436.294,A -85,B 0,C 180,E1 19929.625,E2 19929.625} C_VEL
LIN {X 0,Y 438.055,Z 659.225,A -85,B 0,C 180,E1 19925.818,E2 19925.818} C_VEL
LIN {X 0,Y 437.093,Z 679.388,A -85,B 0,C 180,E1 19925.235,E2 19925.235} C_VEL
LIN {X 0,Y 435.652,Z 698.785,A -85,B 0,C 180,E1 19924.449,E2 19924.449} C_VEL
LIN {X 0,Y 433.835,Z 717.031,A -85,B 0,C 180,E1 19923.49,E2 19923.49} C_VEL
LIN {X 0,Y 432.274,Z 729.797,A -85,B 0,C 180,E1 19922.669,E2 19922.669} C_VEL
LIN {X 0,Y 430.555,Z 736.794,A -85,B 0,C 180,E1 19922.257,E2 19922.257} C_VEL
LIN {X 0,Y 423.097,Z 754.137,A -85,B 0,C 180,E1 19921.338,E2 19921.338} C_VEL
LIN {X 0,Y 421.188,Z 760.526,A -85,B 0,C 180,E1 19920.816,E2 19920.816} C_VEL
LIN {X 0,Y 418.284,Z 776.515,A -85,B 0,C 180,E1 19919.103,E2 19919.103} C_VEL
LIN {X 0,Y 415.237,Z 791.795,A -85,B 0,C 180,E1 19917.145,E2 19917.145} C_VEL
LIN {X 0,Y 412.257,Z 805.93,A -85,B 0,C 180,E1 19914.958,E2 19914.958} C_VEL
LIN {X 0,Y 409.534,Z 818.419,A -85,B 0,C 180,E1 19912.65,E2 19912.65} C_VEL
LIN {X 0,Y 407.083,Z 829.86,A -85,B 0,C 180,E1 19910.11,E2 19910.11} C_VEL
LIN {X 0,Y 405.084,Z 839.498,A -85,B 0,C 180,E1 19907.523,E2 19907.523} C_VEL
LIN {X 0,Y 403.45,Z 848.189,A -85,B 0,C 180,E1 19904.64,E2 19904.64} C_VEL
LIN {X 0,Y 402.227,Z 855.315,A -85,B 0,C 180,E1 19901.614,E2 19901.614} C_VEL
LIN {X 0,Y 401.496,Z 860.561,A -85,B 0,C 180,E1 19898.592,E2 19898.592} C_VEL
LIN {X 0,Y 401.072,Z 864.013,A -85,B 0,C 180,E1 19895.722,E2 19895.722} C_VEL
LIN {X 0,Y 400.87,Z 866.201,A -85,B 0,C 180,E1 19892.572,E2 19892.572} C_VEL
LIN {X 0,Y 400.823,Z 866.773,A -85,B 0,C 180,E1 19889.571,E2 19889.571} C_VEL
LIN {X 0,Y 400.908,Z 865.881,A -85,B 0,C 180,E1 19886.568,E2 19886.568} C_VEL
LIN {X 0,Y 401.186,Z 863.266,A -85,B 0,C 180,E1 19883.417,E2 19883.417} C_VEL
LIN {X 0,Y 401.675,Z 859.133,A -85,B 0,C 180,E1 19880.4,E2 19880.4} C_VEL
LIN {X 0,Y 402.488,Z 853.577,A -85,B 0,C 180,E1 19877.499,E2 19877.499} C_VEL
LIN {X 0,Y 403.832,Z 846.007,A -85,B 0,C 180,E1 19874.491,E2 19874.491} C_VEL
LIN {X 0,Y 405.535,Z 837.323,A -85,B 0,C 180,E1 19871.754,E2 19871.754} C_VEL
LIN {X 0,Y 407.694,Z 827.13,A -85,B 0,C 180,E1 19869.131,E2 19869.131} C_VEL
LIN {X 0,Y 410.286,Z 815.121,A -85,B 0,C 180,E1 19866.597,E2 19866.597} C_VEL
LIN {X 0,Y 413.059,Z 802.144,A -85,B 0,C 180,E1 19864.326,E2 19864.326} C_VEL
LIN {X 0,Y 416.069,Z 787.73,A -85,B 0,C 180,E1 19862.214,E2 19862.214} C_VEL
LIN {X 0,Y 419.186,Z 771.689,A -85,B 0,C 180,E1 19860.254,E2 19860.254} C_VEL
LIN {X 0,Y 422.111,Z 755.373,A -85,B 0,C 180,E1 19858.596,E2 19858.596} C_VEL
LIN {X 0,Y 424.775,Z 738.478,A -85,B 0,C 180,E1 19857.175,E2 19857.175} C_VEL
LIN {X 0,Y 427.077,Z 721.021,A -85,B 0,C 180,E1 19855.973,E2 19855.973} C_VEL
LIN {X 0,Y 429.175,Z 701.746,A -85,B 0,C 180,E1 19854.914,E2 19854.914} C_VEL
LIN {X 0,Y 430.751,Z 682.385,A -85,B 0,C 180,E1 19854.095,E2 19854.095} C_VEL
LIN {X 0,Y 431.819,Z 661.752,A -85,B 0,C 180,E1 19853.471,E2 19853.471} C_VEL
LIN {X 0,Y 432.972,Z 616.471,A -85,B 0,C 180,E1 19852.653,E2 19852.653} C_VEL
LIN {X 0,Y 437.722,Z 439.135,A -85,B 0,C 180,E1 19849.598,E2 19849.598} C_VEL
LIN {X 0,Y 425.827,Z 420.325,A -85,B 0,C 180,E1 19847.626,E2 19847.626} C_VEL
LIN {X 0,Y 415.494,Z 405.504,A -85,B 0,C 180,E1 19845.793,E2 19845.793} C_VEL
LIN {X 0,Y 409.082,Z 396.626,A -85,B 0,C 180,E1 19844.546,E2 19844.546} C_VEL
LIN {X 0,Y 405.508,Z 389.265,A -85,B 0,C 180,E1 19842.886,E2 19842.886} C_VEL
LIN {X 0,Y 403.327,Z 384.89,A -85,B 0,C 180,E1 19841.825,E2 19841.825} C_VEL
LIN {X 0,Y 401.64,Z 381.626,A -85,B 0,C 180,E1 19841.005,E2 19841.005} C_VEL
LIN {X 0,Y 401.486,Z 380.716,A -85,B 0,C 180,E1 19840.58,E2 19840.58} C_VEL
LIN {X 0,Y 401.471,Z 380.7,A -85,B 0,C 180,E1 19836.691,E2 19836.691} C_VEL
LIN {X 0,Y 401.469,Z 380.726,A -85,B 0,C 180,E1 19832.714,E2 19832.714} C_VEL
LIN {X 0,Y 401.464,Z 380.727,A -85,B 0,C 180,E1 19828.73,E2 19828.73} C_VEL
LIN {X 0,Y 401.461,Z 380.725,A -85,B 0,C 180,E1 19824.735,E2 19824.735} C_VEL
LIN {X 0,Y 401.465,Z 380.724,A -85,B 0,C 180,E1 19820.864,E2 19820.864} C_VEL
LIN {X 0,Y 401.479,Z 380.726,A -85,B 0,C 180,E1 19817.012,E2 19817.012} C_VEL
LIN {X 0,Y 401.495,Z 380.72,A -85,B 0,C 180,E1 19813.186,E2 19813.186} C_VEL
LIN {X 0,Y 401.493,Z 380.715,A -85,B 0,C 180,E1 19809.171,E2 19809.171} C_VEL
LIN {X 0,Y 401.478,Z 380.707,A -85,B 0,C 180,E1 19805.287,E2 19805.287} C_VEL
LIN {X 0,Y 401.456,Z 380.707,A -85,B 0,C 180,E1 19801.427,E2 19801.427} C_VEL
LIN {X 0,Y 401.436,Z 380.714,A -85,B 0,C 180,E1 19797.716,E2 19797.716} C_VEL
LIN {X 0,Y 401.432,Z 380.72,A -85,B 0,C 180,E1 19793.852,E2 19793.852} C_VEL
LIN {X 0,Y 401.442,Z 380.724,A -85,B 0,C 180,E1 19790.105,E2 19790.105} C_VEL
LIN {X 0,Y 401.457,Z 380.724,A -85,B 0,C 180,E1 19786.224,E2 19786.224} C_VEL
LIN {X 0,Y 401.468,Z 380.722,A -85,B 0,C 180,E1 19782.312,E2 19782.312} C_VEL
LIN {X 0,Y 401.478,Z 380.709,A -85,B 0,C 180,E1 19778.256,E2 19778.256} C_VEL
LIN {X 0,Y 401.467,Z 380.681,A -85,B 0,C 180,E1 19774.32,E2 19774.32} C_VEL
LIN {X 0,Y 401.441,Z 380.682,A -85,B 0,C 180,E1 19770.616,E2 19770.616} C_VEL
LIN {X 0,Y 401.443,Z 380.791,A -85,B 0,C 180,E1 19768.949,E2 19768.949} C_VEL
LIN {X 0,Y 401.662,Z 381.8,A -85,B 0,C 180,E1 19768.622,E2 19768.622} C_VEL
LIN {X 0,Y 403.646,Z 385.261,A -85,B 0,C 180,E1 19767.821,E2 19767.821} C_VEL
LIN {X 0,Y 406.443,Z 390.243,A -85,B 0,C 180,E1 19766.73,E2 19766.73} C_VEL
LIN {X 0,Y 412.569,Z 401.654,A -85,B 0,C 180,E1 19764.435,E2 19764.435} C_VEL
LIN {X 0,Y 418.967,Z 414.033,A -85,B 0,C 180,E1 19762.17,E2 19762.17} C_VEL
LIN {X 0,Y 426.729,Z 430.281,A -85,B 0,C 180,E1 19759.532,E2 19759.532} C_VEL
LIN {X 0,Y 433.098,Z 444.765,A -85,B 0,C 180,E1 19757.458,E2 19757.458} C_VEL
LIN {X 0,Y 435.593,Z 449.645,A -85,B 0,C 180,E1 19757.027,E2 19757.027} C_VEL
LIN {X 0,Y 439.803,Z 490.73,A -85,B 0,C 180,E1 19755.579,E2 19755.579} C_VEL
LIN {X 0,Y 432.355,Z 713.632,A -85,B 0,C 180,E1 19751.439,E2 19751.439} C_VEL
LIN {X 0,Y 430.94,Z 750.541,A -85,B 0,C 180,E1 19750.708,E2 19750.708} C_VEL
LIN {X 0,Y 429.132,Z 772.86,A -85,B 0,C 180,E1 19750.066,E2 19750.066} C_VEL
LIN {X 0,Y 426.857,Z 794.018,A -85,B 0,C 180,E1 19749.226,E2 19749.226} C_VEL
LIN {X 0,Y 424.254,Z 815.443,A -85,B 0,C 180,E1 19748.127,E2 19748.127} C_VEL
LIN {X 0,Y 421.429,Z 836.31,A -85,B 0,C 180,E1 19746.795,E2 19746.795} C_VEL
LIN {X 0,Y 418.28,Z 857.042,A -85,B 0,C 180,E1 19745.172,E2 19745.172} C_VEL
LIN {X 0,Y 415.241,Z 876.675,A -85,B 0,C 180,E1 19743.329,E2 19743.329} C_VEL
LIN {X 0,Y 412.262,Z 895.364,A -85,B 0,C 180,E1 19741.263,E2 19741.263} C_VEL
LIN {X 0,Y 409.494,Z 913.079,A -85,B 0,C 180,E1 19738.969,E2 19738.969} C_VEL
LIN {X 0,Y 407.091,Z 928.979,A -85,B 0,C 180,E1 19736.55,E2 19736.55} C_VEL
LIN {X 0,Y 404.976,Z 944.049,A -85,B 0,C 180,E1 19733.883,E2 19733.883} C_VEL
LIN {X 0,Y 403.342,Z 956.982,A -85,B 0,C 180,E1 19731.217,E2 19731.217} C_VEL
LIN {X 0,Y 402.125,Z 967.92,A -85,B 0,C 180,E1 19728.557,E2 19728.557} C_VEL
LIN {X 0,Y 401.243,Z 977.53,A -85,B 0,C 180,E1 19725.759,E2 19725.759} C_VEL
LIN {X 0,Y 400.652,Z 985.82,A -85,B 0,C 180,E1 19722.832,E2 19722.832} C_VEL
LIN {X 0,Y 400.351,Z 991.895,A -85,B 0,C 180,E1 19720.068,E2 19720.068} C_VEL
LIN {X 0,Y 400.218,Z 996.721,A -85,B 0,C 180,E1 19717.176,E2 19717.176} C_VEL
LIN {X 0,Y 400.206,Z 999.729,A -85,B 0,C 180,E1 19714.442,E2 19714.442} C_VEL
LIN {X 0,Y 400.209,Z 1001.435,A -85,B 0,C 180,E1 19711.432,E2 19711.432} C_VEL
LIN {X 0,Y 400.21,Z 1001.488,A -85,B 0,C 180,E1 19708.855,E2 19708.855} C_VEL
LIN {X 0,Y 400.205,Z 999.983,A -85,B 0,C 180,E1 19705.846,E2 19705.846} C_VEL
LIN {X 0,Y 400.228,Z 997.084,A -85,B 0,C 180,E1 19703.114,E2 19703.114} C_VEL
LIN {X 0,Y 400.321,Z 992.468,A -85,B 0,C 180,E1 19700.223,E2 19700.223} C_VEL
LIN {X 0,Y 400.611,Z 986.516,A -85,B 0,C 180,E1 19697.461,E2 19697.461} C_VEL
LIN {X 0,Y 401.168,Z 978.455,A -85,B 0,C 180,E1 19694.535,E2 19694.535} C_VEL
LIN {X 0,Y 402.014,Z 969.075,A -85,B 0,C 180,E1 19691.74,E2 19691.74} C_VEL
LIN {X 0,Y 403.264,Z 957.643,A -85,B 0,C 180,E1 19688.932,E2 19688.932} C_VEL
LIN {X 0,Y 404.977,Z 944.063,A -85,B 0,C 180,E1 19686.118,E2 19686.118} C_VEL
LIN {X 0,Y 407.091,Z 928.99,A -85,B 0,C 180,E1 19683.451,E2 19683.451} C_VEL
LIN {X 0,Y 409.598,Z 912.444,A -85,B 0,C 180,E1 19680.941,E2 19680.941} C_VEL
LIN {X 0,Y 412.31,Z 895.06,A -85,B 0,C 180,E1 19678.7,E2 19678.7} C_VEL
LIN {X 0,Y 415.244,Z 876.663,A -85,B 0,C 180,E1 19676.671,E2 19676.671} C_VEL
LIN {X 0,Y 418.278,Z 857.045,A -85,B 0,C 180,E1 19674.829,E2 19674.829} C_VEL
LIN {X 0,Y 421.284,Z 837.218,A -85,B 0,C 180,E1 19673.272,E2 19673.272} C_VEL
LIN {X 0,Y 424.079,Z 816.719,A -85,B 0,C 180,E1 19671.95,E2 19671.95} C_VEL
LIN {X 0,Y 426.767,Z 794.755,A -85,B 0,C 180,E1 19670.808,E2 19670.808} C_VEL
LIN {X 0,Y 429.114,Z 772.958,A -85,B 0,C 180,E1 19669.939,E2 19669.939} C_VEL
LIN {X 0,Y 430.921,Z 750.635,A -85,B 0,C 180,E1 19669.297,E2 19669.297} C_VEL
LIN {X 0,Y 432.339,Z 713.667,A -85,B 0,C 180,E1 19668.564,E2 19668.564} C_VEL
LIN {X 0,Y 439.77,Z 491.04,A -85,B 0,C 180,E1 19664.43,E2 19664.43} C_VEL
LIN {X 0,Y 439.203,Z 483.875,A -85,B 0,C 180,E1 19664.202,E2 19664.202} C_VEL
LIN {X 0,Y 435.292,Z 448.762,A -85,B 0,C 180,E1 19662.926,E2 19662.926} C_VEL
LIN {X 0,Y 432.364,Z 443.306,A -85,B 0,C 180,E1 19662.384,E2 19662.384} C_VEL
LIN {X 0,Y 424.357,Z 425.111,A -85,B 0,C 180,E1 19659.681,E2 19659.681} C_VEL
LIN {X 0,Y 417.403,Z 410.967,A -85,B 0,C 180,E1 19657.303,E2 19657.303} C_VEL
LIN {X 0,Y 411.066,Z 398.78,A -85,B 0,C 180,E1 19655.032,E2 19655.032} C_VEL
LIN {X 0,Y 406.39,Z 390.177,A -85,B 0,C 180,E1 19653.274,E2 19653.274} C_VEL
LIN {X 0,Y 404.312,Z 386.372,A -85,B 0,C 180,E1 19652.455,E2 19652.455} C_VEL
LIN {X 0,Y 401.828,Z 382.319,A -85,B 0,C 180,E1 19651.502,E2 19651.502} C_VEL
LIN {X 0,Y 401.446,Z 380.801,A -85,B 0,C 180,E1 19651.072,E2 19651.072} C_VEL
LIN {X 0,Y 401.456,Z 380.731,A -85,B 0,C 180,E1 19647.436,E2 19647.436} C_VEL
LIN {X 0,Y 401.456,Z 380.669,A -85,B 0,C 180,E1 19643.484,E2 19643.484} C_VEL
LIN {X 0,Y 401.472,Z 380.714,A -85,B 0,C 180,E1 19639.646,E2 19639.646} C_VEL
LIN {X 0,Y 401.471,Z 380.711,A -85,B 0,C 180,E1 19635.603,E2 19635.603} C_VEL
LIN {X 0,Y 401.447,Z 380.714,A -85,B 0,C 180,E1 19631.784,E2 19631.784} C_VEL
LIN {X 0,Y 401.43,Z 380.72,A -85,B 0,C 180,E1 19628.018,E2 19628.018} C_VEL
LIN {X 0,Y 401.432,Z 380.726,A -85,B 0,C 180,E1 19624.142,E2 19624.142} C_VEL
LIN {X 0,Y 401.435,Z 380.73,A -85,B 0,C 180,E1 19620.142,E2 19620.142} C_VEL
LIN {X 0,Y 401.444,Z 380.728,A -85,B 0,C 180,E1 19616.287,E2 19616.287} C_VEL
LIN {X 0,Y 401.461,Z 380.721,A -85,B 0,C 180,E1 19612.415,E2 19612.415} C_VEL
LIN {X 0,Y 401.477,Z 380.711,A -85,B 0,C 180,E1 19608.507,E2 19608.507} C_VEL
LIN {X 0,Y 401.496,Z 380.707,A -85,B 0,C 180,E1 19604.546,E2 19604.546} C_VEL
LIN {X 0,Y 401.495,Z 380.707,A -85,B 0,C 180,E1 19600.506,E2 19600.506} C_VEL
LIN {X 0,Y 401.485,Z 380.708,A -85,B 0,C 180,E1 19596.673,E2 19596.673} C_VEL
LIN {X 0,Y 401.477,Z 380.709,A -85,B 0,C 180,E1 19592.726,E2 19592.726} C_VEL
LIN {X 0,Y 401.462,Z 380.712,A -85,B 0,C 180,E1 19588.943,E2 19588.943} C_VEL
LIN {X 0,Y 401.463,Z 380.72,A -85,B 0,C 180,E1 19585.014,E2 19585.014} C_VEL
LIN {X 0,Y 401.46,Z 380.67,A -85,B 0,C 180,E1 19580.984,E2 19580.984} C_VEL
LIN {X 0,Y 401.496,Z 380.918,A -85,B 0,C 180,E1 19579.083,E2 19579.083} C_VEL
LIN {X 0,Y 402.731,Z 384.114,A -85,B 0,C 180,E1 19578.289,E2 19578.289} C_VEL
LIN {X 0,Y 404.017,Z 386.259,A -85,B 0,C 180,E1 19577.721,E2 19577.721} C_VEL
LIN {X 0,Y 408.552,Z 395.517,A -85,B 0,C 180,E1 19575.578,E2 19575.578} C_VEL
LIN {X 0,Y 410.135,Z 398.111,A -85,B 0,C 180,E1 19575.108,E2 19575.108} C_VEL
LIN {X 0,Y 420.989,Z 413.271,A -85,B 0,C 180,E1 19573.111,E2 19573.111} C_VEL
LIN {X 0,Y 432.913,Z 431.336,A -85,B 0,C 180,E1 19571.079,E2 19571.079} C_VEL
LIN {X 0,Y 437.789,Z 439.636,A -85,B 0,C 180,E1 19570.282,E2 19570.282} C_VEL
LIN {X 0,Y 431.841,Z 660.123,A -85,B 0,C 180,E1 19566.472,E2 19566.472} C_VEL
LIN {X 0,Y 430.842,Z 680.269,A -85,B 0,C 180,E1 19565.884,E2 19565.884} C_VEL
LIN {X 0,Y 429.308,Z 700.057,A -85,B 0,C 180,E1 19565.073,E2 19565.073} C_VEL
LIN {X 0,Y 427.373,Z 718.55,A -85,B 0,C 180,E1 19564.085,E2 19564.085} C_VEL
LIN {X 0,Y 424.975,Z 737.016,A -85,B 0,C 180,E1 19562.845,E2 19562.845} C_VEL
LIN {X 0,Y 422.237,Z 754.452,A -85,B 0,C 180,E1 19561.393,E2 19561.393} C_VEL
LIN {X 0,Y 421.188,Z 760.526,A -85,B 0,C 180,E1 19560.816,E2 19560.816} C_VEL
LIN {X 0,Y 419.256,Z 766.921,A -85,B 0,C 180,E1 19560.263,E2 19560.263} C_VEL
LIN {X 0,Y 411.266,Z 782.798,A -85,B 0,C 180,E1 19558.964,E2 19558.964} C_VEL
LIN {X 0,Y 409.246,Z 788.514,A -85,B 0,C 180,E1 19558.299,E2 19558.299} C_VEL
LIN {X 0,Y 406.264,Z 802.201,A -85,B 0,C 180,E1 19556.292,E2 19556.292} C_VEL
LIN {X 0,Y 403.31,Z 815.351,A -85,B 0,C 180,E1 19553.987,E2 19553.987} C_VEL
LIN {X 0,Y 400.613,Z 827.028,A -85,B 0,C 180,E1 19551.521,E2 19551.521} C_VEL
LIN {X 0,Y 398.243,Z 837.598,A -85,B 0,C 180,E1 19548.821,E2 19548.821} C_VEL
LIN {X 0,Y 396.311,Z 846.709,A -85,B 0,C 180,E1 19545.96,E2 19545.96} C_VEL
LIN {X 0,Y 394.895,Z 854.151,A -85,B 0,C 180,E1 19543.021,E2 19543.021} C_VEL
LIN {X 0,Y 393.932,Z 860.021,A -85,B 0,C 180,E1 19540,E2 19540} C_VEL
LIN {X 0,Y 393.365,Z 864.353,A -85,B 0,C 180,E1 19536.86,E2 19536.86} C_VEL
LIN {X 0,Y 393.045,Z 866.948,A -85,B 0,C 180,E1 19533.791,E2 19533.791} C_VEL
LIN {X 0,Y 392.942,Z 868.046,A -85,B 0,C 180,E1 19530.728,E2 19530.728} C_VEL
LIN {X 0,Y 392.978,Z 867.63,A -85,B 0,C 180,E1 19527.521,E2 19527.521} C_VEL
LIN {X 0,Y 393.178,Z 865.725,A -85,B 0,C 180,E1 19524.455,E2 19524.455} C_VEL
LIN {X 0,Y 393.636,Z 862.279,A -85,B 0,C 180,E1 19521.381,E2 19521.381} C_VEL
LIN {X 0,Y 394.44,Z 856.856,A -85,B 0,C 180,E1 19518.152,E2 19518.152} C_VEL
LIN {X 0,Y 395.737,Z 849.791,A -85,B 0,C 180,E1 19515.067,E2 19515.067} C_VEL
LIN {X 0,Y 397.367,Z 841.643,A -85,B 0,C 180,E1 19512.276,E2 19512.276} C_VEL
LIN {X 0,Y 399.58,Z 831.622,A -85,B 0,C 180,E1 19509.495,E2 19509.495} C_VEL
LIN {X 0,Y 402.199,Z 820.104,A -85,B 0,C 180,E1 19506.874,E2 19506.874} C_VEL
LIN {X 0,Y 405.017,Z 807.905,A -85,B 0,C 180,E1 19504.563,E2 19504.563} C_VEL
LIN {X 0,Y 408.238,Z 793.372,A -85,B 0,C 180,E1 19502.27,E2 19502.27} C_VEL
LIN {X 0,Y 411.425,Z 778.133,A -85,B 0,C 180,E1 19500.282,E2 19500.282} C_VEL
LIN {X 0,Y 414.514,Z 761.968,A -85,B 0,C 180,E1 19498.521,E2 19498.521} C_VEL
LIN {X 0,Y 417.57,Z 744.111,A -85,B 0,C 180,E1 19496.914,E2 19496.914} C_VEL
LIN {X 0,Y 420.201,Z 726.145,A -85,B 0,C 180,E1 19495.592,E2 19495.592} C_VEL
LIN {X 0,Y 422.452,Z 707.416,A -85,B 0,C 180,E1 19494.488,E2 19494.488} C_VEL
LIN {X 0,Y 424.211,Z 687.826,A -85,B 0,C 180,E1 19493.602,E2 19493.602} C_VEL
LIN {X 0,Y 425.431,Z 667.691,A -85,B 0,C 180,E1 19492.936,E2 19492.936} C_VEL
LIN {X 0,Y 426.173,Z 643.62,A -85,B 0,C 180,E1 19492.421,E2 19492.421} C_VEL
LIN {X 0,Y 431.87,Z 442.603,A -85,B 0,C 180,E1 19488.928,E2 19488.928} C_VEL
LIN {X 0,Y 420.827,Z 425.117,A -85,B 0,C 180,E1 19487.037,E2 19487.037} C_VEL
LIN {X 0,Y 409.447,Z 408.605,A -85,B 0,C 180,E1 19484.938,E2 19484.938} C_VEL
LIN {X 0,Y 401.215,Z 397.458,A -85,B 0,C 180,E1 19483.261,E2 19483.261} C_VEL
LIN {X 0,Y 397.739,Z 390.451,A -85,B 0,C 180,E1 19481.58,E2 19481.58} C_VEL
LIN {X 0,Y 395.285,Z 385.727,A -85,B 0,C 180,E1 19480.357,E2 19480.357} C_VEL
LIN {X 0,Y 393.573,Z 381.966,A -85,B 0,C 180,E1 19479.335,E2 19479.335} C_VEL
LIN {X 0,Y 393.532,Z 381.673,A -85,B 0,C 180,E1 19477.207,E2 19477.207} C_VEL
LIN {X 0,Y 393.54,Z 381.704,A -85,B 0,C 180,E1 19473.284,E2 19473.284} C_VEL
LIN {X 0,Y 393.549,Z 381.708,A -85,B 0,C 180,E1 19469.363,E2 19469.363} C_VEL
LIN {X 0,Y 393.555,Z 381.709,A -85,B 0,C 180,E1 19465.427,E2 19465.427} C_VEL
LIN {X 0,Y 393.567,Z 381.707,A -85,B 0,C 180,E1 19461.459,E2 19461.459} C_VEL
LIN {X 0,Y 393.559,Z 381.708,A -85,B 0,C 180,E1 19457.445,E2 19457.445} C_VEL
LIN {X 0,Y 393.55,Z 381.706,A -85,B 0,C 180,E1 19453.518,E2 19453.518} C_VEL
LIN {X 0,Y 393.535,Z 381.701,A -85,B 0,C 180,E1 19449.506,E2 19449.506} C_VEL
LIN {X 0,Y 393.511,Z 381.696,A -85,B 0,C 180,E1 19445.687,E2 19445.687} C_VEL
LIN {X 0,Y 393.503,Z 381.697,A -85,B 0,C 180,E1 19441.748,E2 19441.748} C_VEL
LIN {X 0,Y 393.496,Z 381.703,A -85,B 0,C 180,E1 19437.816,E2 19437.816} C_VEL
LIN {X 0,Y 393.494,Z 381.708,A -85,B 0,C 180,E1 19433.874,E2 19433.874} C_VEL
LIN {X 0,Y 393.5,Z 381.713,A -85,B 0,C 180,E1 19430.051,E2 19430.051} C_VEL
LIN {X 0,Y 393.515,Z 381.713,A -85,B 0,C 180,E1 19426.182,E2 19426.182} C_VEL
LIN {X 0,Y 393.524,Z 381.711,A -85,B 0,C 180,E1 19422.249,E2 19422.249} C_VEL
LIN {X 0,Y 393.54,Z 381.694,A -85,B 0,C 180,E1 19418.227,E2 19418.227} C_VEL
LIN {X 0,Y 393.53,Z 381.668,A -85,B 0,C 180,E1 19414.249,E2 19414.249} C_VEL
LIN {X 0,Y 393.556,Z 381.917,A -85,B 0,C 180,E1 19410.371,E2 19410.371} C_VEL
LIN {X 0,Y 394.514,Z 384.651,A -85,B 0,C 180,E1 19409.712,E2 19409.712} C_VEL
LIN {X 0,Y 396.362,Z 387.081,A -85,B 0,C 180,E1 19409.029,E2 19409.029} C_VEL
LIN {X 0,Y 398.285,Z 390.865,A -85,B 0,C 180,E1 19408.185,E2 19408.185} C_VEL
LIN {X 0,Y 399.625,Z 393.384,A -85,B 0,C 180,E1 19407.628,E2 19407.628} C_VEL
LIN {X 0,Y 402.455,Z 398.393,A -85,B 0,C 180,E1 19406.528,E2 19406.528} C_VEL
LIN {X 0,Y 408.656,Z 409.766,A -85,B 0,C 180,E1 19404.214,E2 19404.214} C_VEL
LIN {X 0,Y 416.502,Z 425.694,A -85,B 0,C 180,E1 19401.38,E2 19401.38} C_VEL
LIN {X 0,Y 424.442,Z 443.33,A -85,B 0,C 180,E1 19398.642,E2 19398.642} C_VEL
LIN {X 0,Y 430.043,Z 453.441,A -85,B 0,C 180,E1 19397.649,E2 19397.649} C_VEL
LIN {X 0,Y 433.858,Z 491.983,A -85,B 0,C 180,E1 19396.268,E2 19396.268} C_VEL
LIN {X 0,Y 426.012,Z 715.553,A -85,B 0,C 180,E1 19392.068,E2 19392.068} C_VEL
LIN {X 0,Y 424.594,Z 750.01,A -85,B 0,C 180,E1 19391.37,E2 19391.37} C_VEL
LIN {X 0,Y 422.682,Z 772.577,A -85,B 0,C 180,E1 19390.711,E2 19390.711} C_VEL
LIN {X 0,Y 420.224,Z 794.157,A -85,B 0,C 180,E1 19389.835,E2 19389.835} C_VEL
LIN {X 0,Y 417.412,Z 815.847,A -85,B 0,C 180,E1 19388.692,E2 19388.692} C_VEL
LIN {X 0,Y 414.476,Z 836.281,A -85,B 0,C 180,E1 19387.354,E2 19387.354} C_VEL
LIN {X 0,Y 411.297,Z 856.112,A -85,B 0,C 180,E1 19385.775,E2 19385.775} C_VEL
LIN {X 0,Y 408.162,Z 875.24,A -85,B 0,C 180,E1 19383.95,E2 19383.95} C_VEL
LIN {X 0,Y 404.951,Z 894.215,A -85,B 0,C 180,E1 19381.819,E2 19381.819} C_VEL
LIN {X 0,Y 402.046,Z 911.808,A -85,B 0,C 180,E1 19379.497,E2 19379.497} C_VEL
LIN {X 0,Y 399.406,Z 928.244,A -85,B 0,C 180,E1 19376.941,E2 19376.941} C_VEL
LIN {X 0,Y 397.267,Z 942.542,A -85,B 0,C 180,E1 19374.343,E2 19374.343} C_VEL
LIN {X 0,Y 395.472,Z 955.958,A -85,B 0,C 180,E1 19371.503,E2 19371.503} C_VEL
LIN {X 0,Y 394.152,Z 967.451,A -85,B 0,C 180,E1 19368.639,E2 19368.639} C_VEL
LIN {X 0,Y 393.268,Z 976.905,A -85,B 0,C 180,E1 19365.785,E2 19365.785} C_VEL
LIN {X 0,Y 392.692,Z 985.047,A -85,B 0,C 180,E1 19362.794,E2 19362.794} C_VEL
LIN {X 0,Y 392.422,Z 990.757,A -85,B 0,C 180,E1 19360.125,E2 19360.125} C_VEL
LIN {X 0,Y 392.303,Z 995.53,A -85,B 0,C 180,E1 19357.174,E2 19357.174} C_VEL
LIN {X 0,Y 392.303,Z 998.38,A -85,B 0,C 180,E1 19354.532,E2 19354.532} C_VEL
LIN {X 0,Y 392.316,Z 1000.077,A -85,B 0,C 180,E1 19351.607,E2 19351.607} C_VEL
LIN {X 0,Y 392.318,Z 1000.185,A -85,B 0,C 180,E1 19348.978,E2 19348.978} C_VEL
LIN {X 0,Y 392.304,Z 998.891,A -85,B 0,C 180,E1 19346.055,E2 19346.055} C_VEL
LIN {X 0,Y 392.318,Z 996.083,A -85,B 0,C 180,E1 19343.269,E2 19343.269} C_VEL
LIN {X 0,Y 392.379,Z 991.622,A -85,B 0,C 180,E1 19340.319,E2 19340.319} C_VEL
LIN {X 0,Y 392.652,Z 985.741,A -85,B 0,C 180,E1 19337.501,E2 19337.501} C_VEL
LIN {X 0,Y 393.192,Z 977.832,A -85,B 0,C 180,E1 19334.516,E2 19334.516} C_VEL
LIN {X 0,Y 394.059,Z 968.363,A -85,B 0,C 180,E1 19331.614,E2 19331.614} C_VEL
LIN {X 0,Y 395.314,Z 957.247,A -85,B 0,C 180,E1 19328.799,E2 19328.799} C_VEL
LIN {X 0,Y 397.18,Z 943.165,A -85,B 0,C 180,E1 19325.777,E2 19325.777} C_VEL
LIN {X 0,Y 399.264,Z 929.175,A -85,B 0,C 180,E1 19323.211,E2 19323.211} C_VEL
LIN {X 0,Y 401.866,Z 912.82,A -85,B 0,C 180,E1 19320.654,E2 19320.654} C_VEL
LIN {X 0,Y 404.735,Z 895.477,A -85,B 0,C 180,E1 19318.339,E2 19318.339} C_VEL
LIN {X 0,Y 408.03,Z 876.02,A -85,B 0,C 180,E1 19316.131,E2 19316.131} C_VEL
LIN {X 0,Y 411.163,Z 856.962,A -85,B 0,C 180,E1 19314.299,E2 19314.299} C_VEL
LIN {X 0,Y 414.307,Z 837.28,A -85,B 0,C 180,E1 19312.722,E2 19312.722} C_VEL
LIN {X 0,Y 417.276,Z 816.765,A -85,B 0,C 180,E1 19311.365,E2 19311.365} C_VEL
LIN {X 0,Y 420.031,Z 795.707,A -85,B 0,C 180,E1 19310.237,E2 19310.237} C_VEL
LIN {X 0,Y 422.547,Z 773.757,A -85,B 0,C 180,E1 19309.332,E2 19309.332} C_VEL
LIN {X 0,Y 424.478,Z 751.358,A -85,B 0,C 180,E1 19308.668,E2 19308.668} C_VEL
LIN {X 0,Y 425.833,Z 720.326,A -85,B 0,C 180,E1 19308.025,E2 19308.025} C_VEL
LIN {X 0,Y 433.68,Z 496.057,A -85,B 0,C 180,E1 19303.812,E2 19303.812} C_VEL
LIN {X 0,Y 433.699,Z 489.138,A -85,B 0,C 180,E1 19303.655,E2 19303.655} C_VEL
LIN {X 0,Y 429.789,Z 452.748,A -85,B 0,C 180,E1 19302.314,E2 19302.314} C_VEL
LIN {X 0,Y 424.143,Z 442.786,A -85,B 0,C 180,E1 19301.304,E2 19301.304} C_VEL
LIN {X 0,Y 416.462,Z 425.647,A -85,B 0,C 180,E1 19298.624,E2 19298.624} C_VEL
LIN {X 0,Y 408.615,Z 409.702,A -85,B 0,C 180,E1 19295.79,E2 19295.79} C_VEL
LIN {X 0,Y 401.408,Z 396.26,A -85,B 0,C 180,E1 19293.059,E2 19293.059} C_VEL
LIN {X 0,Y 398.248,Z 390.806,A -85,B 0,C 180,E1 19291.818,E2 19291.818} C_VEL
LIN {X 0,Y 395.941,Z 386.517,A -85,B 0,C 180,E1 19290.839,E2 19290.839} C_VEL
LIN {X 0,Y 393.897,Z 383.213,A -85,B 0,C 180,E1 19290.004,E2 19290.004} C_VEL
LIN {X 0,Y 393.527,Z 381.748,A -85,B 0,C 180,E1 19289.563,E2 19289.563} C_VEL
LIN {X 0,Y 393.53,Z 381.667,A -85,B 0,C 180,E1 19285.751,E2 19285.751} C_VEL
LIN {X 0,Y 393.539,Z 381.693,A -85,B 0,C 180,E1 19281.773,E2 19281.773} C_VEL
LIN {X 0,Y 393.529,Z 381.711,A -85,B 0,C 180,E1 19277.697,E2 19277.697} C_VEL
LIN {X 0,Y 393.526,Z 381.713,A -85,B 0,C 180,E1 19273.667,E2 19273.667} C_VEL
LIN {X 0,Y 393.517,Z 381.713,A -85,B 0,C 180,E1 19269.653,E2 19269.653} C_VEL
LIN {X 0,Y 393.5,Z 381.712,A -85,B 0,C 180,E1 19265.833,E2 19265.833} C_VEL
LIN {X 0,Y 393.498,Z 381.705,A -85,B 0,C 180,E1 19261.893,E2 19261.893} C_VEL
LIN {X 0,Y 393.495,Z 381.698,A -85,B 0,C 180,E1 19257.961,E2 19257.961} C_VEL
LIN {X 0,Y 393.499,Z 381.695,A -85,B 0,C 180,E1 19254.02,E2 19254.02} C_VEL
LIN {X 0,Y 393.513,Z 381.698,A -85,B 0,C 180,E1 19250.198,E2 19250.198} C_VEL
LIN {X 0,Y 393.535,Z 381.705,A -85,B 0,C 180,E1 19246.332,E2 19246.332} C_VEL
LIN {X 0,Y 393.549,Z 381.709,A -85,B 0,C 180,E1 19242.402,E2 19242.402} C_VEL
LIN {X 0,Y 393.568,Z 381.708,A -85,B 0,C 180,E1 19238.384,E2 19238.384} C_VEL
LIN {X 0,Y 393.559,Z 381.708,A -85,B 0,C 180,E1 19234.395,E2 19234.395} C_VEL
LIN {X 0,Y 393.555,Z 381.705,A -85,B 0,C 180,E1 19230.47,E2 19230.47} C_VEL
LIN {X 0,Y 393.543,Z 381.703,A -85,B 0,C 180,E1 19226.542,E2 19226.542} C_VEL
LIN {X 0,Y 393.531,Z 381.67,A -85,B 0,C 180,E1 19222.61,E2 19222.61} C_VEL
LIN {X 0,Y 393.57,Z 381.944,A -85,B 0,C 180,E1 19220.554,E2 19220.554} C_VEL
LIN {X 0,Y 395.091,Z 385.482,A -85,B 0,C 180,E1 19219.61,E2 19219.61} C_VEL
LIN {X 0,Y 396.063,Z 387.032,A -85,B 0,C 180,E1 19219.168,E2 19219.168} C_VEL
LIN {X 0,Y 398.093,Z 390.88,A -85,B 0,C 180,E1 19218.176,E2 19218.176} C_VEL
LIN {X 0,Y 401.767,Z 398.336,A -85,B 0,C 180,E1 19216.47,E2 19216.47} C_VEL
LIN {X 0,Y 413.624,Z 414.495,A -85,B 0,C 180,E1 19214.165,E2 19214.165} C_VEL
LIN {X 0,Y 425.57,Z 432.468,A -85,B 0,C 180,E1 19212.03,E2 19212.03} C_VEL
LIN {X 0,Y 431.911,Z 443.006,A -85,B 0,C 180,E1 19210.956,E2 19210.956} C_VEL
LIN {X 0,Y 425.679,Z 661.1,A -85,B 0,C 180,E1 19207.143,E2 19207.143} C_VEL
LIN {X 0,Y 424.631,Z 681.378,A -85,B 0,C 180,E1 19206.544,E2 19206.544} C_VEL
LIN {X 0,Y 423.014,Z 701.312,A -85,B 0,C 180,E1 19205.715,E2 19205.715} C_VEL
LIN {X 0,Y 420.898,Z 720.483,A -85,B 0,C 180,E1 19204.672,E2 19204.672} C_VEL
LIN {X 0,Y 418.408,Z 738.773,A -85,B 0,C 180,E1 19203.419,E2 19203.419} C_VEL
LIN {X 0,Y 415.566,Z 756.054,A -85,B 0,C 180,E1 19201.956,E2 19201.956} C_VEL
LIN {X 0,Y 412.501,Z 772.498,A -85,B 0,C 180,E1 19200.272,E2 19200.272} C_VEL
LIN {X 0,Y 409.246,Z 788.514,A -85,B 0,C 180,E1 19198.299,E2 19198.299} C_VEL
LIN {X 0,Y 407.226,Z 794.179,A -85,B 0,C 180,E1 19197.604,E2 19197.604} C_VEL
LIN {X 0,Y 398.966,Z 808.244,A -85,B 0,C 180,E1 19195.927,E2 19195.927} C_VEL
LIN {X 0,Y 396.934,Z 813.183,A -85,B 0,C 180,E1 19195.125,E2 19195.125} C_VEL
LIN {X 0,Y 394.027,Z 825.209,A -85,B 0,C 180,E1 19192.685,E2 19192.685} C_VEL
LIN {X 0,Y 391.45,Z 836.117,A -85,B 0,C 180,E1 19190.012,E2 19190.012} C_VEL
LIN {X 0,Y 389.167,Z 845.999,A -85,B 0,C 180,E1 19187.029,E2 19187.029} C_VEL
LIN {X 0,Y 387.512,Z 853.846,A -85,B 0,C 180,E1 19184.032,E2 19184.032} C_VEL
LIN {X 0,Y 386.36,Z 859.923,A -85,B 0,C 180,E1 19181.039,E2 19181.039} C_VEL
LIN {X 0,Y 385.642,Z 864.603,A -85,B 0,C 180,E1 19177.897,E2 19177.897} C_VEL
LIN {X 0,Y 385.239,Z 867.684,A -85,B 0,C 180,E1 19174.763,E2 19174.763} C_VEL
LIN {X 0,Y 385.066,Z 869.262,A -85,B 0,C 180,E1 19171.636,E2 19171.636} C_VEL
LIN {X 0,Y 385.056,Z 869.293,A -85,B 0,C 180,E1 19168.512,E2 19168.512} C_VEL
LIN {X 0,Y 385.219,Z 867.822,A -85,B 0,C 180,E1 19165.344,E2 19165.344} C_VEL
LIN {X 0,Y 385.626,Z 864.721,A -85,B 0,C 180,E1 19162.102,E2 19162.102} C_VEL
LIN {X 0,Y 386.337,Z 860.091,A -85,B 0,C 180,E1 19158.959,E2 19158.959} C_VEL
LIN {X 0,Y 387.474,Z 854.068,A -85,B 0,C 180,E1 19155.963,E2 19155.963} C_VEL
LIN {X 0,Y 389.163,Z 846.06,A -85,B 0,C 180,E1 19152.895,E2 19152.895} C_VEL
LIN {X 0,Y 391.375,Z 836.437,A -85,B 0,C 180,E1 19149.982,E2 19149.982} C_VEL
LIN {X 0,Y 393.941,Z 825.6,A -85,B 0,C 180,E1 19147.309,E2 19147.309} C_VEL
LIN {X 0,Y 396.917,Z 813.326,A -85,B 0,C 180,E1 19144.806,E2 19144.806} C_VEL
LIN {X 0,Y 400.162,Z 799.579,A -85,B 0,C 180,E1 19142.47,E2 19142.47} C_VEL
LIN {X 0,Y 403.388,Z 785.375,A -85,B 0,C 180,E1 19140.448,E2 19140.448} C_VEL
LIN {X 0,Y 406.749,Z 769.254,A -85,B 0,C 180,E1 19138.538,E2 19138.538} C_VEL
LIN {X 0,Y 409.894,Z 752.332,A -85,B 0,C 180,E1 19136.882,E2 19136.882} C_VEL
LIN {X 0,Y 412.83,Z 734.308,A -85,B 0,C 180,E1 19135.434,E2 19135.434} C_VEL
LIN {X 0,Y 415.39,Z 715.391,A -85,B 0,C 180,E1 19134.207,E2 19134.207} C_VEL
LIN {X 0,Y 417.424,Z 696.142,A -85,B 0,C 180,E1 19133.223,E2 19133.223} C_VEL
LIN {X 0,Y 418.981,Z 675.548,A -85,B 0,C 180,E1 19132.445,E2 19132.445} C_VEL
LIN {X 0,Y 419.818,Z 655.362,A -85,B 0,C 180,E1 19131.929,E2 19131.929} C_VEL
LIN {X 0,Y 426.083,Z 446.015,A -85,B 0,C 180,E1 19128.24,E2 19128.24} C_VEL
LIN {X 0,Y 414.353,Z 427.585,A -85,B 0,C 180,E1 19126.154,E2 19126.154} C_VEL
LIN {X 0,Y 404.059,Z 412.757,A -85,B 0,C 180,E1 19124.178,E2 19124.178} C_VEL
LIN {X 0,Y 394.341,Z 399.871,A -85,B 0,C 180,E1 19122.166,E2 19122.166} C_VEL
LIN {X 0,Y 393.152,Z 397.869,A -85,B 0,C 180,E1 19121.784,E2 19121.784} C_VEL
LIN {X 0,Y 389.767,Z 391.297,A -85,B 0,C 180,E1 19120.082,E2 19120.082} C_VEL
LIN {X 0,Y 387.399,Z 386.798,A -85,B 0,C 180,E1 19118.842,E2 19118.842} C_VEL
LIN {X 0,Y 385.669,Z 383.01,A -85,B 0,C 180,E1 19117.754,E2 19117.754} C_VEL
LIN {X 0,Y 385.596,Z 382.675,A -85,B 0,C 180,E1 19116.613,E2 19116.613} C_VEL
LIN {X 0,Y 385.595,Z 382.705,A -85,B 0,C 180,E1 19112.578,E2 19112.578} C_VEL
LIN {X 0,Y 385.587,Z 382.705,A -85,B 0,C 180,E1 19108.668,E2 19108.668} C_VEL
LIN {X 0,Y 385.583,Z 382.703,A -85,B 0,C 180,E1 19104.677,E2 19104.677} C_VEL
LIN {X 0,Y 385.58,Z 382.701,A -85,B 0,C 180,E1 19100.604,E2 19100.604} C_VEL
LIN {X 0,Y 385.578,Z 382.703,A -85,B 0,C 180,E1 19096.574,E2 19096.574} C_VEL
LIN {X 0,Y 385.586,Z 382.707,A -85,B 0,C 180,E1 19092.734,E2 19092.734} C_VEL
LIN {X 0,Y 385.596,Z 382.7,A -85,B 0,C 180,E1 19088.8,E2 19088.8} C_VEL
LIN {X 0,Y 385.603,Z 382.689,A -85,B 0,C 180,E1 19084.909,E2 19084.909} C_VEL
LIN {X 0,Y 385.611,Z 382.683,A -85,B 0,C 180,E1 19080.892,E2 19080.892} C_VEL
LIN {X 0,Y 385.597,Z 382.684,A -85,B 0,C 180,E1 19076.879,E2 19076.879} C_VEL
LIN {X 0,Y 385.598,Z 382.684,A -85,B 0,C 180,E1 19072.851,E2 19072.851} C_VEL
LIN {X 0,Y 385.584,Z 382.686,A -85,B 0,C 180,E1 19068.786,E2 19068.786} C_VEL
LIN {X 0,Y 385.572,Z 382.689,A -85,B 0,C 180,E1 19064.817,E2 19064.817} C_VEL
LIN {X 0,Y 385.556,Z 382.692,A -85,B 0,C 180,E1 19060.928,E2 19060.928} C_VEL
LIN {X 0,Y 385.546,Z 382.655,A -85,B 0,C 180,E1 19057.108,E2 19057.108} C_VEL
LIN {X 0,Y 385.552,Z 382.694,A -85,B 0,C 180,E1 19053.128,E2 19053.128} C_VEL
LIN {X 0,Y 385.64,Z 382.989,A -85,B 0,C 180,E1 19051.971,E2 19051.971} C_VEL
LIN {X 0,Y 387.008,Z 386.37,A -85,B 0,C 180,E1 19051.111,E2 19051.111} C_VEL
LIN {X 0,Y 388.518,Z 388.019,A -85,B 0,C 180,E1 19050.558,E2 19050.558} C_VEL
LIN {X 0,Y 390.357,Z 391.857,A -85,B 0,C 180,E1 19049.668,E2 19049.668} C_VEL
LIN {X 0,Y 391.663,Z 393.975,A -85,B 0,C 180,E1 19049.128,E2 19049.128} C_VEL
LIN {X 0,Y 394.652,Z 399.488,A -85,B 0,C 180,E1 19047.857,E2 19047.857} C_VEL
LIN {X 0,Y 399.243,Z 407.711,A -85,B 0,C 180,E1 19046.05,E2 19046.05} C_VEL
LIN {X 0,Y 406.083,Z 421.132,A -85,B 0,C 180,E1 19043.427,E2 19043.427} C_VEL
LIN {X 0,Y 413.207,Z 435.994,A -85,B 0,C 180,E1 19040.835,E2 19040.835} C_VEL
LIN {X 0,Y 416.305,Z 442.769,A -85,B 0,C 180,E1 19039.795,E2 19039.795} C_VEL
LIN {X 0,Y 424.543,Z 457.176,A -85,B 0,C 180,E1 19038.289,E2 19038.289} C_VEL
LIN {X 0,Y 427.972,Z 493.361,A -85,B 0,C 180,E1 19036.974,E2 19036.974} C_VEL
LIN {X 0,Y 419.757,Z 716.606,A -85,B 0,C 180,E1 19032.733,E2 19032.733} C_VEL
LIN {X 0,Y 418.319,Z 749.353,A -85,B 0,C 180,E1 19032.057,E2 19032.057} C_VEL
LIN {X 0,Y 416.323,Z 771.963,A -85,B 0,C 180,E1 19031.387,E2 19031.387} C_VEL
LIN {X 0,Y 413.737,Z 793.57,A -85,B 0,C 180,E1 19030.498,E2 19030.498} C_VEL
LIN {X 0,Y 410.781,Z 815.111,A -85,B 0,C 180,E1 19029.347,E2 19029.347} C_VEL
LIN {X 0,Y 407.688,Z 835.503,A -85,B 0,C 180,E1 19027.99,E2 19027.99} C_VEL
LIN {X 0,Y 404.231,Z 856.065,A -85,B 0,C 180,E1 19026.324,E2 19026.324} C_VEL
LIN {X 0,Y 400.936,Z 874.97,A -85,B 0,C 180,E1 19024.475,E2 19024.475} C_VEL
LIN {X 0,Y 397.447,Z 894.423,A -85,B 0,C 180,E1 19022.228,E2 19022.228} C_VEL
LIN {X 0,Y 394.455,Z 911.524,A -85,B 0,C 180,E1 19019.901,E2 19019.901} C_VEL
LIN {X 0,Y 391.738,Z 927.56,A -85,B 0,C 180,E1 19017.348,E2 19017.348} C_VEL
LIN {X 0,Y 389.454,Z 941.956,A -85,B 0,C 180,E1 19014.656,E2 19014.656} C_VEL
LIN {X 0,Y 387.525,Z 955.665,A -85,B 0,C 180,E1 19011.65,E2 19011.65} C_VEL
LIN {X 0,Y 386.18,Z 966.959,A -85,B 0,C 180,E1 19008.725,E2 19008.725} C_VEL
LIN {X 0,Y 385.292,Z 976.288,A -85,B 0,C 180,E1 19005.811,E2 19005.811} C_VEL
LIN {X 0,Y 384.733,Z 984.265,A -85,B 0,C 180,E1 19002.761,E2 19002.761} C_VEL
LIN {X 0,Y 384.46,Z 990.204,A -85,B 0,C 180,E1 18999.883,E2 18999.883} C_VEL
LIN {X 0,Y 384.403,Z 994.706,A -85,B 0,C 180,E1 18996.872,E2 18996.872} C_VEL
LIN {X 0,Y 384.405,Z 997.548,A -85,B 0,C 180,E1 18994.027,E2 18994.027} C_VEL
LIN {X 0,Y 384.431,Z 998.855,A -85,B 0,C 180,E1 18991.044,E2 18991.044} C_VEL
LIN {X 0,Y 384.422,Z 998.718,A -85,B 0,C 180,E1 18988.212,E2 18988.212} C_VEL
LIN {X 0,Y 384.396,Z 996.906,A -85,B 0,C 180,E1 18985.226,E2 18985.226} C_VEL
LIN {X 0,Y 384.383,Z 993.724,A -85,B 0,C 180,E1 18982.329,E2 18982.329} C_VEL
LIN {X 0,Y 384.534,Z 988.774,A -85,B 0,C 180,E1 18979.363,E2 18979.363} C_VEL
LIN {X 0,Y 384.866,Z 982.086,A -85,B 0,C 180,E1 18976.318,E2 18976.318} C_VEL
LIN {X 0,Y 385.493,Z 974.001,A -85,B 0,C 180,E1 18973.425,E2 18973.425} C_VEL
LIN {X 0,Y 386.572,Z 963.371,A -85,B 0,C 180,E1 18970.3,E2 18970.3} C_VEL
LIN {X 0,Y 388.046,Z 951.745,A -85,B 0,C 180,E1 18967.426,E2 18967.426} C_VEL
LIN {X 0,Y 389.985,Z 938.487,A -85,B 0,C 180,E1 18964.652,E2 18964.652} C_VEL
LIN {X 0,Y 392.33,Z 923.873,A -85,B 0,C 180,E1 18962.039,E2 18962.039} C_VEL
LIN {X 0,Y 395.141,Z 907.481,A -85,B 0,C 180,E1 18959.517,E2 18959.517} C_VEL
LIN {X 0,Y 398.343,Z 889.632,A -85,B 0,C 180,E1 18957.173,E2 18957.173} C_VEL
LIN {X 0,Y 401.689,Z 870.699,A -85,B 0,C 180,E1 18955.08,E2 18955.08} C_VEL
LIN {X 0,Y 404.951,Z 851.788,A -85,B 0,C 180,E1 18953.313,E2 18953.313} C_VEL
LIN {X 0,Y 408.295,Z 831.47,A -85,B 0,C 180,E1 18951.721,E2 18951.721} C_VEL
LIN {X 0,Y 411.473,Z 810.489,A -85,B 0,C 180,E1 18950.38,E2 18950.38} C_VEL
LIN {X 0,Y 414.213,Z 789.751,A -85,B 0,C 180,E1 18949.332,E2 18949.332} C_VEL
LIN {X 0,Y 416.758,Z 767.196,A -85,B 0,C 180,E1 18948.461,E2 18948.461} C_VEL
LIN {X 0,Y 418.596,Z 744.835,A -85,B 0,C 180,E1 18947.835,E2 18947.835} C_VEL
LIN {X 0,Y 425.865,Z 548.924,A -85,B 0,C 180,E1 18944.081,E2 18944.081} C_VEL
LIN {X 0,Y 427.857,Z 490.811,A -85,B 0,C 180,E1 18942.96,E2 18942.96} C_VEL
LIN {X 0,Y 424.265,Z 456.537,A -85,B 0,C 180,E1 18941.673,E2 18941.673} C_VEL
LIN {X 0,Y 415.83,Z 441.957,A -85,B 0,C 180,E1 18940.12,E2 18940.12} C_VEL
LIN {X 0,Y 408.27,Z 425.591,A -85,B 0,C 180,E1 18937.398,E2 18937.398} C_VEL
LIN {X 0,Y 400.977,Z 410.892,A -85,B 0,C 180,E1 18934.636,E2 18934.636} C_VEL
LIN {X 0,Y 395.659,Z 401.277,A -85,B 0,C 180,E1 18932.565,E2 18932.565} C_VEL
LIN {X 0,Y 393.308,Z 396.883,A -85,B 0,C 180,E1 18931.58,E2 18931.58} C_VEL
LIN {X 0,Y 390.626,Z 392.189,A -85,B 0,C 180,E1 18930.451,E2 18930.451} C_VEL
LIN {X 0,Y 388.61,Z 388.258,A -85,B 0,C 180,E1 18929.519,E2 18929.519} C_VEL
LIN {X 0,Y 386.042,Z 384.574,A -85,B 0,C 180,E1 18928.461,E2 18928.461} C_VEL
LIN {X 0,Y 385.619,Z 382.823,A -85,B 0,C 180,E1 18927.989,E2 18927.989} C_VEL
LIN {X 0,Y 385.588,Z 382.637,A -85,B 0,C 180,E1 18923.861,E2 18923.861} C_VEL
LIN {X 0,Y 385.584,Z 382.694,A -85,B 0,C 180,E1 18919.858,E2 18919.858} C_VEL
LIN {X 0,Y 385.571,Z 382.692,A -85,B 0,C 180,E1 18915.853,E2 18915.853} C_VEL
LIN {X 0,Y 385.557,Z 382.693,A -85,B 0,C 180,E1 18911.973,E2 18911.973} C_VEL
LIN {X 0,Y 385.551,Z 382.696,A -85,B 0,C 180,E1 18908.05,E2 18908.05} C_VEL
LIN {X 0,Y 385.554,Z 382.702,A -85,B 0,C 180,E1 18904.164,E2 18904.164} C_VEL
LIN {X 0,Y 385.557,Z 382.708,A -85,B 0,C 180,E1 18900.148,E2 18900.148} C_VEL
LIN {X 0,Y 385.563,Z 382.706,A -85,B 0,C 180,E1 18896.134,E2 18896.134} C_VEL
LIN {X 0,Y 385.574,Z 382.701,A -85,B 0,C 180,E1 18892.25,E2 18892.25} C_VEL
LIN {X 0,Y 385.587,Z 382.692,A -85,B 0,C 180,E1 18888.33,E2 18888.33} C_VEL
LIN {X 0,Y 385.614,Z 382.684,A -85,B 0,C 180,E1 18884.51,E2 18884.51} C_VEL
LIN {X 0,Y 385.616,Z 382.683,A -85,B 0,C 180,E1 18880.459,E2 18880.459} C_VEL
LIN {X 0,Y 385.619,Z 382.683,A -85,B 0,C 180,E1 18876.465,E2 18876.465} C_VEL
LIN {X 0,Y 385.623,Z 382.685,A -85,B 0,C 180,E1 18872.346,E2 18872.346} C_VEL
LIN {X 0,Y 385.615,Z 382.69,A -85,B 0,C 180,E1 18868.415,E2 18868.415} C_VEL
LIN {X 0,Y 385.604,Z 382.702,A -85,B 0,C 180,E1 18864.491,E2 18864.491} C_VEL
LIN {X 0,Y 385.662,Z 382.959,A -85,B 0,C 180,E1 18862.147,E2 18862.147} C_VEL
LIN {X 0,Y 387.188,Z 386.542,A -85,B 0,C 180,E1 18861.133,E2 18861.133} C_VEL
LIN {X 0,Y 388.361,Z 388.477,A -85,B 0,C 180,E1 18860.559,E2 18860.559} C_VEL
LIN {X 0,Y 390.815,Z 393.31,A -85,B 0,C 180,E1 18859.278,E2 18859.278} C_VEL
LIN {X 0,Y 393.454,Z 398.539,A -85,B 0,C 180,E1 18857.962,E2 18857.962} C_VEL
LIN {X 0,Y 403.001,Z 411.231,A -85,B 0,C 180,E1 18855.923,E2 18855.923} C_VEL
LIN {X 0,Y 415.098,Z 428.663,A -85,B 0,C 180,E1 18853.603,E2 18853.603} C_VEL
LIN {X 0,Y 426.101,Z 446.136,A -85,B 0,C 180,E1 18851.653,E2 18851.653} C_VEL
LIN {X 0,Y 419.577,Z 662.049,A -85,B 0,C 180,E1 18847.834,E2 18847.834} C_VEL
LIN {X 0,Y 418.494,Z 682.194,A -85,B 0,C 180,E1 18847.233,E2 18847.233} C_VEL
LIN {X 0,Y 416.846,Z 701.826,A -85,B 0,C 180,E1 18846.412,E2 18846.412} C_VEL
LIN {X 0,Y 414.747,Z 720.415,A -85,B 0,C 180,E1 18845.402,E2 18845.402} C_VEL
LIN {X 0,Y 412.039,Z 739.528,A -85,B 0,C 180,E1 18844.089,E2 18844.089} C_VEL
LIN {X 0,Y 408.935,Z 757.643,A -85,B 0,C 180,E1 18842.537,E2 18842.537} C_VEL
LIN {X 0,Y 405.735,Z 774.02,A -85,B 0,C 180,E1 18840.832,E2 18840.832} C_VEL
LIN {X 0,Y 402.312,Z 790.057,A -85,B 0,C 180,E1 18838.822,E2 18838.822} C_VEL
LIN {X 0,Y 398.989,Z 804.506,A -85,B 0,C 180,E1 18836.649,E2 18836.649} C_VEL
LIN {X 0,Y 396.934,Z 813.183,A -85,B 0,C 180,E1 18835.125,E2 18835.125} C_VEL
LIN {X 0,Y 394.917,Z 818.052,A -85,B 0,C 180,E1 18834.291,E2 18834.291} C_VEL
LIN {X 0,Y 386.734,Z 830.025,A -85,B 0,C 180,E1 18832.247,E2 18832.247} C_VEL
LIN {X 0,Y 384.827,Z 834.103,A -85,B 0,C 180,E1 18831.314,E2 18831.314} C_VEL
LIN {X 0,Y 382.342,Z 844.108,A -85,B 0,C 180,E1 18828.444,E2 18828.444} C_VEL
LIN {X 0,Y 380.469,Z 852.289,A -85,B 0,C 180,E1 18825.546,E2 18825.546} C_VEL
LIN {X 0,Y 378.964,Z 859.387,A -85,B 0,C 180,E1 18822.338,E2 18822.338} C_VEL
LIN {X 0,Y 378,Z 864.828,A -85,B 0,C 180,E1 18818.977,E2 18818.977} C_VEL
LIN {X 0,Y 377.454,Z 868.304,A -85,B 0,C 180,E1 18815.776,E2 18815.776} C_VEL
LIN {X 0,Y 377.213,Z 870.25,A -85,B 0,C 180,E1 18812.582,E2 18812.582} C_VEL
LIN {X 0,Y 377.162,Z 870.716,A -85,B 0,C 180,E1 18809.24,E2 18809.24} C_VEL
LIN {X 0,Y 377.287,Z 869.677,A -85,B 0,C 180,E1 18806.049,E2 18806.049} C_VEL
LIN {X 0,Y 377.657,Z 867.136,A -85,B 0,C 180,E1 18802.852,E2 18802.852} C_VEL
LIN {X 0,Y 378.296,Z 862.95,A -85,B 0,C 180,E1 18799.647,E2 18799.647} C_VEL
LIN {X 0,Y 379.379,Z 857.264,A -85,B 0,C 180,E1 18796.534,E2 18796.534} C_VEL
LIN {X 0,Y 381.028,Z 849.707,A -85,B 0,C 180,E1 18793.381,E2 18793.381} C_VEL
LIN {X 0,Y 383.26,Z 840.433,A -85,B 0,C 180,E1 18790.335,E2 18790.335} C_VEL
LIN {X 0,Y 385.838,Z 830.223,A -85,B 0,C 180,E1 18787.61,E2 18787.61} C_VEL
LIN {X 0,Y 388.819,Z 818.638,A -85,B 0,C 180,E1 18785.058,E2 18785.058} C_VEL
LIN {X 0,Y 392.062,Z 805.585,A -85,B 0,C 180,E1 18782.677,E2 18782.677} C_VEL
LIN {X 0,Y 395.556,Z 791.09,A -85,B 0,C 180,E1 18780.471,E2 18780.471} C_VEL
LIN {X 0,Y 399.146,Z 775.002,A -85,B 0,C 180,E1 18778.433,E2 18778.433} C_VEL
LIN {X 0,Y 402.49,Z 758.561,A -85,B 0,C 180,E1 18776.704,E2 18776.704} C_VEL
LIN {X 0,Y 405.693,Z 740.67,A -85,B 0,C 180,E1 18775.156,E2 18775.156} C_VEL
LIN {X 0,Y 408.46,Z 721.942,A -85,B 0,C 180,E1 18773.851,E2 18773.851} C_VEL
LIN {X 0,Y 410.68,Z 703.224,A -85,B 0,C 180,E1 18772.818,E2 18772.818} C_VEL
LIN {X 0,Y 412.455,Z 682.916,A -85,B 0,C 180,E1 18771.96,E2 18771.96} C_VEL
LIN {X 0,Y 413.579,Z 662.803,A -85,B 0,C 180,E1 18771.356,E2 18771.356} C_VEL
LIN {X 0,Y 420.274,Z 449.402,A -85,B 0,C 180,E1 18767.52,E2 18767.52} C_VEL
LIN {X 0,Y 409.108,Z 431.864,A -85,B 0,C 180,E1 18765.463,E2 18765.463} C_VEL
LIN {X 0,Y 398.75,Z 416.845,A -85,B 0,C 180,E1 18763.397,E2 18763.397} C_VEL
LIN {X 0,Y 388.037,Z 402.634,A -85,B 0,C 180,E1 18761.076,E2 18761.076} C_VEL
LIN {X 0,Y 385.515,Z 399.232,A -85,B 0,C 180,E1 18760.421,E2 18760.421} C_VEL
LIN {X 0,Y 382.291,Z 392.869,A -85,B 0,C 180,E1 18758.689,E2 18758.689} C_VEL
LIN {X 0,Y 379.713,Z 388.083,A -85,B 0,C 180,E1 18757.275,E2 18757.275} C_VEL
LIN {X 0,Y 378.001,Z 385.157,A -85,B 0,C 180,E1 18756.336,E2 18756.336} C_VEL
LIN {X 0,Y 377.689,Z 383.719,A -85,B 0,C 180,E1 18755.807,E2 18755.807} C_VEL
LIN {X 0,Y 377.687,Z 383.682,A -85,B 0,C 180,E1 18751.791,E2 18751.791} C_VEL
LIN {X 0,Y 377.689,Z 383.675,A -85,B 0,C 180,E1 18747.771,E2 18747.771} C_VEL
LIN {X 0,Y 377.681,Z 383.671,A -85,B 0,C 180,E1 18743.665,E2 18743.665} C_VEL
LIN {X 0,Y 377.673,Z 383.671,A -85,B 0,C 180,E1 18739.647,E2 18739.647} C_VEL
LIN {X 0,Y 377.663,Z 383.675,A -85,B 0,C 180,E1 18735.667,E2 18735.667} C_VEL
LIN {X 0,Y 377.645,Z 383.684,A -85,B 0,C 180,E1 18731.763,E2 18731.763} C_VEL
LIN {X 0,Y 377.639,Z 383.692,A -85,B 0,C 180,E1 18727.761,E2 18727.761} C_VEL
LIN {X 0,Y 377.629,Z 383.695,A -85,B 0,C 180,E1 18723.796,E2 18723.796} C_VEL
LIN {X 0,Y 377.623,Z 383.696,A -85,B 0,C 180,E1 18719.849,E2 18719.849} C_VEL
LIN {X 0,Y 377.618,Z 383.691,A -85,B 0,C 180,E1 18715.749,E2 18715.749} C_VEL
LIN {X 0,Y 377.614,Z 383.689,A -85,B 0,C 180,E1 18711.627,E2 18711.627} C_VEL
LIN {X 0,Y 377.611,Z 383.688,A -85,B 0,C 180,E1 18707.616,E2 18707.616} C_VEL
LIN {X 0,Y 377.608,Z 383.691,A -85,B 0,C 180,E1 18703.542,E2 18703.542} C_VEL
LIN {X 0,Y 377.612,Z 383.697,A -85,B 0,C 180,E1 18699.543,E2 18699.543} C_VEL
LIN {X 0,Y 377.614,Z 383.629,A -85,B 0,C 180,E1 18695.603,E2 18695.603} C_VEL
LIN {X 0,Y 377.676,Z 383.959,A -85,B 0,C 180,E1 18693.761,E2 18693.761} C_VEL
LIN {X 0,Y 379.008,Z 387.297,A -85,B 0,C 180,E1 18692.846,E2 18692.846} C_VEL
LIN {X 0,Y 380.746,Z 389.412,A -85,B 0,C 180,E1 18692.132,E2 18692.132} C_VEL
LIN {X 0,Y 382.484,Z 392.916,A -85,B 0,C 180,E1 18691.25,E2 18691.25} C_VEL
LIN {X 0,Y 383.85,Z 394.888,A -85,B 0,C 180,E1 18690.679,E2 18690.679} C_VEL
LIN {X 0,Y 389.062,Z 404.234,A -85,B 0,C 180,E1 18688.382,E2 18688.382} C_VEL
LIN {X 0,Y 395.978,Z 417.171,A -85,B 0,C 180,E1 18685.556,E2 18685.556} C_VEL
LIN {X 0,Y 403.554,Z 432.514,A -85,B 0,C 180,E1 18682.626,E2 18682.626} C_VEL
LIN {X 0,Y 407.935,Z 441.852,A -85,B 0,C 180,E1 18681.07,E2 18681.07} C_VEL
LIN {X 0,Y 419.092,Z 460.886,A -85,B 0,C 180,E1 18678.947,E2 18678.947} C_VEL
LIN {X 0,Y 422.157,Z 494.625,A -85,B 0,C 180,E1 18677.701,E2 18677.701} C_VEL
LIN {X 0,Y 413.538,Z 718.312,A -85,B 0,C 180,E1 18673.406,E2 18673.406} C_VEL
LIN {X 0,Y 412.068,Z 749.207,A -85,B 0,C 180,E1 18672.751,E2 18672.751} C_VEL
LIN {X 0,Y 410.001,Z 771.514,A -85,B 0,C 180,E1 18672.078,E2 18672.078} C_VEL
LIN {X 0,Y 407.32,Z 792.941,A -85,B 0,C 180,E1 18671.184,E2 18671.184} C_VEL
LIN {X 0,Y 404.214,Z 814.397,A -85,B 0,C 180,E1 18670.022,E2 18670.022} C_VEL
LIN {X 0,Y 400.981,Z 834.583,A -85,B 0,C 180,E1 18668.66,E2 18668.66} C_VEL
LIN {X 0,Y 397.356,Z 855.189,A -85,B 0,C 180,E1 18666.966,E2 18666.966} C_VEL
LIN {X 0,Y 393.821,Z 874.315,A -85,B 0,C 180,E1 18665.062,E2 18665.062} C_VEL
LIN {X 0,Y 390.33,Z 892.805,A -85,B 0,C 180,E1 18662.889,E2 18662.889} C_VEL
LIN {X 0,Y 387.098,Z 910.117,A -85,B 0,C 180,E1 18660.498,E2 18660.498} C_VEL
LIN {X 0,Y 384.241,Z 925.983,A -85,B 0,C 180,E1 18657.927,E2 18657.927} C_VEL
LIN {X 0,Y 381.87,Z 940.024,A -85,B 0,C 180,E1 18655.262,E2 18655.262} C_VEL
LIN {X 0,Y 379.838,Z 953.503,A -85,B 0,C 180,E1 18652.273,E2 18652.273} C_VEL
LIN {X 0,Y 378.384,Z 964.929,A -85,B 0,C 180,E1 18649.286,E2 18649.286} C_VEL
LIN {X 0,Y 377.391,Z 974.8,A -85,B 0,C 180,E1 18646.151,E2 18646.151} C_VEL
LIN {X 0,Y 376.793,Z 983.159,A -85,B 0,C 180,E1 18642.879,E2 18642.879} C_VEL
LIN {X 0,Y 376.524,Z 989.195,A -85,B 0,C 180,E1 18639.876,E2 18639.876} C_VEL
LIN {X 0,Y 376.487,Z 993.523,A -85,B 0,C 180,E1 18636.864,E2 18636.864} C_VEL
LIN {X 0,Y 376.506,Z 996.327,A -85,B 0,C 180,E1 18633.959,E2 18633.959} C_VEL
LIN {X 0,Y 376.542,Z 997.527,A -85,B 0,C 180,E1 18631.065,E2 18631.065} C_VEL
LIN {X 0,Y 376.531,Z 997.388,A -85,B 0,C 180,E1 18628.175,E2 18628.175} C_VEL
LIN {X 0,Y 376.495,Z 995.685,A -85,B 0,C 180,E1 18625.279,E2 18625.279} C_VEL
LIN {X 0,Y 376.466,Z 992.78,A -85,B 0,C 180,E1 18622.524,E2 18622.524} C_VEL
LIN {X 0,Y 376.589,Z 987.927,A -85,B 0,C 180,E1 18619.446,E2 18619.446} C_VEL
LIN {X 0,Y 376.895,Z 981.424,A -85,B 0,C 180,E1 18616.345,E2 18616.345} C_VEL
LIN {X 0,Y 377.557,Z 972.973,A -85,B 0,C 180,E1 18613.225,E2 18613.225} C_VEL
LIN {X 0,Y 378.668,Z 962.504,A -85,B 0,C 180,E1 18610.051,E2 18610.051} C_VEL
LIN {X 0,Y 380.215,Z 950.91,A -85,B 0,C 180,E1 18607.098,E2 18607.098} C_VEL
LIN {X 0,Y 382.246,Z 937.711,A -85,B 0,C 180,E1 18604.268,E2 18604.268} C_VEL
LIN {X 0,Y 384.716,Z 923.218,A -85,B 0,C 180,E1 18601.605,E2 18601.605} C_VEL
LIN {X 0,Y 387.669,Z 906.963,A -85,B 0,C 180,E1 18599.037,E2 18599.037} C_VEL
LIN {X 0,Y 391.023,Z 889.219,A -85,B 0,C 180,E1 18596.654,E2 18596.654} C_VEL
LIN {X 0,Y 394.533,Z 870.446,A -85,B 0,C 180,E1 18594.53,E2 18594.53} C_VEL
LIN {X 0,Y 398.108,Z 850.906,A -85,B 0,C 180,E1 18592.666,E2 18592.666} C_VEL
LIN {X 0,Y 401.537,Z 831.145,A -85,B 0,C 180,E1 18591.088,E2 18591.088} C_VEL
LIN {X 0,Y 404.955,Z 809.681,A -85,B 0,C 180,E1 18589.698,E2 18589.698} C_VEL
LIN {X 0,Y 407.801,Z 789.174,A -85,B 0,C 180,E1 18588.647,E2 18588.647} C_VEL
LIN {X 0,Y 410.448,Z 766.843,A -85,B 0,C 180,E1 18587.77,E2 18587.77} C_VEL
LIN {X 0,Y 412.392,Z 744.41,A -85,B 0,C 180,E1 18587.129,E2 18587.129} C_VEL
LIN {X 0,Y 419.833,Z 553.191,A -85,B 0,C 180,E1 18583.423,E2 18583.423} C_VEL
LIN {X 0,Y 422.041,Z 492.12,A -85,B 0,C 180,E1 18582.233,E2 18582.233} C_VEL
LIN {X 0,Y 418.799,Z 460.305,A -85,B 0,C 180,E1 18581.014,E2 18581.014} C_VEL
LIN {X 0,Y 407.205,Z 440.522,A -85,B 0,C 180,E1 18578.765,E2 18578.765} C_VEL
LIN {X 0,Y 399.5,Z 424.186,A -85,B 0,C 180,E1 18575.848,E2 18575.848} C_VEL
LIN {X 0,Y 392.391,Z 410.507,A -85,B 0,C 180,E1 18573.044,E2 18573.044} C_VEL
LIN {X 0,Y 387.629,Z 401.85,A -85,B 0,C 180,E1 18571.056,E2 18571.056} C_VEL
LIN {X 0,Y 385.692,Z 398.259,A -85,B 0,C 180,E1 18570.193,E2 18570.193} C_VEL
LIN {X 0,Y 383.147,Z 393.696,A -85,B 0,C 180,E1 18569.037,E2 18569.037} C_VEL
LIN {X 0,Y 381.175,Z 390.65,A -85,B 0,C 180,E1 18568.174,E2 18568.174} C_VEL
LIN {X 0,Y 380.383,Z 388.766,A -85,B 0,C 180,E1 18567.726,E2 18567.726} C_VEL
LIN {X 0,Y 378.349,Z 386.169,A -85,B 0,C 180,E1 18566.865,E2 18566.865} C_VEL
LIN {X 0,Y 377.665,Z 383.897,A -85,B 0,C 180,E1 18566.239,E2 18566.239} C_VEL
LIN {X 0,Y 377.612,Z 383.65,A -85,B 0,C 180,E1 18562.413,E2 18562.413} C_VEL
LIN {X 0,Y 377.608,Z 383.683,A -85,B 0,C 180,E1 18558.526,E2 18558.526} C_VEL
LIN {X 0,Y 377.605,Z 383.685,A -85,B 0,C 180,E1 18554.412,E2 18554.412} C_VEL
LIN {X 0,Y 377.61,Z 383.684,A -85,B 0,C 180,E1 18550.373,E2 18550.373} C_VEL
LIN {X 0,Y 377.612,Z 383.683,A -85,B 0,C 180,E1 18546.232,E2 18546.232} C_VEL
LIN {X 0,Y 377.616,Z 383.679,A -85,B 0,C 180,E1 18542.124,E2 18542.124} C_VEL
LIN {X 0,Y 377.618,Z 383.674,A -85,B 0,C 180,E1 18538.027,E2 18538.027} C_VEL
LIN {X 0,Y 377.621,Z 383.671,A -85,B 0,C 180,E1 18533.92,E2 18533.92} C_VEL
LIN {X 0,Y 377.626,Z 383.673,A -85,B 0,C 180,E1 18529.781,E2 18529.781} C_VEL
LIN {X 0,Y 377.628,Z 383.677,A -85,B 0,C 180,E1 18525.688,E2 18525.688} C_VEL
LIN {X 0,Y 377.634,Z 383.68,A -85,B 0,C 180,E1 18521.634,E2 18521.634} C_VEL
LIN {X 0,Y 377.638,Z 383.68,A -85,B 0,C 180,E1 18517.588,E2 18517.588} C_VEL
LIN {X 0,Y 377.645,Z 383.678,A -85,B 0,C 180,E1 18513.589,E2 18513.589} C_VEL
LIN {X 0,Y 377.653,Z 383.676,A -85,B 0,C 180,E1 18509.656,E2 18509.656} C_VEL
LIN {X 0,Y 377.664,Z 383.677,A -85,B 0,C 180,E1 18505.673,E2 18505.673} C_VEL
LIN {X 0,Y 377.722,Z 383.985,A -85,B 0,C 180,E1 18503.876,E2 18503.876} C_VEL
LIN {X 0,Y 379.153,Z 387.421,A -85,B 0,C 180,E1 18502.85,E2 18502.85} C_VEL
LIN {X 0,Y 380.424,Z 389.2,A -85,B 0,C 180,E1 18502.237,E2 18502.237} C_VEL
LIN {X 0,Y 382.421,Z 393.042,A -85,B 0,C 180,E1 18501.134,E2 18501.134} C_VEL
LIN {X 0,Y 385.832,Z 399.866,A -85,B 0,C 180,E1 18499.326,E2 18499.326} C_VEL
LIN {X 0,Y 396.036,Z 413.167,A -85,B 0,C 180,E1 18497.055,E2 18497.055} C_VEL
LIN {X 0,Y 407.806,Z 429.822,A -85,B 0,C 180,E1 18494.682,E2 18494.682} C_VEL
LIN {X 0,Y 420.039,Z 449.073,A -85,B 0,C 180,E1 18492.417,E2 18492.417} C_VEL
LIN {X 0,Y 420.322,Z 450.26,A -85,B 0,C 180,E1 18492.35,E2 18492.35} C_VEL
LIN {X 0,Y 413.536,Z 662.974,A -85,B 0,C 180,E1 18488.545,E2 18488.545} C_VEL
LIN {X 0,Y 412.403,Z 683.201,A -85,B 0,C 180,E1 18487.934,E2 18487.934} C_VEL
LIN {X 0,Y 410.664,Z 703.052,A -85,B 0,C 180,E1 18487.095,E2 18487.095} C_VEL
LIN {X 0,Y 408.45,Z 721.793,A -85,B 0,C 180,E1 18486.062,E2 18486.062} C_VEL
LIN {X 0,Y 405.725,Z 740.254,A -85,B 0,C 180,E1 18484.781,E2 18484.781} C_VEL
LIN {X 0,Y 402.62,Z 757.673,A -85,B 0,C 180,E1 18483.282,E2 18483.282} C_VEL
LIN {X 0,Y 399.277,Z 774.265,A -85,B 0,C 180,E1 18481.555,E2 18481.555} C_VEL
LIN {X 0,Y 395.672,Z 790.478,A -85,B 0,C 180,E1 18479.518,E2 18479.518} C_VEL
LIN {X 0,Y 392.402,Z 804.208,A -85,B 0,C 180,E1 18477.461,E2 18477.461} C_VEL
LIN {X 0,Y 389.103,Z 817.418,A -85,B 0,C 180,E1 18475.084,E2 18475.084} C_VEL
LIN {X 0,Y 386.072,Z 829.191,A -85,B 0,C 180,E1 18472.535,E2 18472.535} C_VEL
LIN {X 0,Y 384.827,Z 834.103,A -85,B 0,C 180,E1 18471.314,E2 18471.314} C_VEL
LIN {X 0,Y 382.96,Z 838.08,A -85,B 0,C 180,E1 18470.353,E2 18470.353} C_VEL
LIN {X 0,Y 375.135,Z 847.784,A -85,B 0,C 180,E1 18467.963,E2 18467.963} C_VEL
LIN {X 0,Y 373.444,Z 850.955,A -85,B 0,C 180,E1 18466.913,E2 18466.913} C_VEL
LIN {X 0,Y 371.677,Z 858.537,A -85,B 0,C 180,E1 18463.692,E2 18463.692} C_VEL
LIN {X 0,Y 370.525,Z 864.155,A -85,B 0,C 180,E1 18460.572,E2 18460.572} C_VEL
LIN {X 0,Y 369.82,Z 868.371,A -85,B 0,C 180,E1 18457.299,E2 18457.299} C_VEL
LIN {X 0,Y 369.414,Z 870.944,A -85,B 0,C 180,E1 18454.034,E2 18454.034} C_VEL
LIN {X 0,Y 369.277,Z 872.031,A -85,B 0,C 180,E1 18450.775,E2 18450.775} C_VEL
LIN {X 0,Y 369.323,Z 871.618,A -85,B 0,C 180,E1 18447.362,E2 18447.362} C_VEL
LIN {X 0,Y 369.585,Z 869.73,A -85,B 0,C 180,E1 18444.099,E2 18444.099} C_VEL
LIN {X 0,Y 370.168,Z 866.306,A -85,B 0,C 180,E1 18440.83,E2 18440.83} C_VEL
LIN {X 0,Y 371.189,Z 860.905,A -85,B 0,C 180,E1 18437.398,E2 18437.398} C_VEL
LIN {X 0,Y 372.69,Z 854.236,A -85,B 0,C 180,E1 18434.279,E2 18434.279} C_VEL
LIN {X 0,Y 374.64,Z 846.23,A -85,B 0,C 180,E1 18431.323,E2 18431.323} C_VEL
LIN {X 0,Y 377.238,Z 836.369,A -85,B 0,C 180,E1 18428.384,E2 18428.384} C_VEL
LIN {X 0,Y 380.111,Z 825.75,A -85,B 0,C 180,E1 18425.775,E2 18425.775} C_VEL
LIN {X 0,Y 383.527,Z 813.003,A -85,B 0,C 180,E1 18423.194,E2 18423.194} C_VEL
LIN {X 0,Y 386.949,Z 799.607,A -85,B 0,C 180,E1 18420.939,E2 18420.939} C_VEL
LIN {X 0,Y 390.691,Z 784.301,A -85,B 0,C 180,E1 18418.789,E2 18418.789} C_VEL
LIN {X 0,Y 394.322,Z 767.973,A -85,B 0,C 180,E1 18416.881,E2 18416.881} C_VEL
LIN {X 0,Y 397.676,Z 751.275,A -85,B 0,C 180,E1 18415.262,E2 18415.262} C_VEL
LIN {X 0,Y 400.744,Z 733.311,A -85,B 0,C 180,E1 18413.842,E2 18413.842} C_VEL
LIN {X 0,Y 403.281,Z 715.259,A -85,B 0,C 180,E1 18412.689,E2 18412.689} C_VEL
LIN {X 0,Y 405.507,Z 694.881,A -85,B 0,C 180,E1 18411.67,E2 18411.67} C_VEL
LIN {X 0,Y 407.066,Z 674.88,A -85,B 0,C 180,E1 18410.933,E2 18410.933} C_VEL
LIN {X 0,Y 407.935,Z 654.465,A -85,B 0,C 180,E1 18410.422,E2 18410.422} C_VEL
LIN {X 0,Y 414.641,Z 452.934,A -85,B 0,C 180,E1 18406.8,E2 18406.8} C_VEL
LIN {X 0,Y 402.946,Z 434.594,A -85,B 0,C 180,E1 18404.557,E2 18404.557} C_VEL
LIN {X 0,Y 391.751,Z 418.557,A -85,B 0,C 180,E1 18402.213,E2 18402.213} C_VEL
LIN {X 0,Y 380.528,Z 403.912,A -85,B 0,C 180,E1 18399.631,E2 18399.631} C_VEL
LIN {X 0,Y 377.77,Z 400.129,A -85,B 0,C 180,E1 18398.85,E2 18398.85} C_VEL
LIN {X 0,Y 374.54,Z 394.058,A -85,B 0,C 180,E1 18397.048,E2 18397.048} C_VEL
LIN {X 0,Y 372.587,Z 390.256,A -85,B 0,C 180,E1 18395.869,E2 18395.869} C_VEL
LIN {X 0,Y 370.201,Z 386.585,A -85,B 0,C 180,E1 18394.545,E2 18394.545} C_VEL
LIN {X 0,Y 369.782,Z 384.932,A -85,B 0,C 180,E1 18394.036,E2 18394.036} C_VEL
LIN {X 0,Y 369.742,Z 384.663,A -85,B 0,C 180,E1 18390.019,E2 18390.019} C_VEL
LIN {X 0,Y 369.73,Z 384.667,A -85,B 0,C 180,E1 18385.983,E2 18385.983} C_VEL
LIN {X 0,Y 369.726,Z 384.669,A -85,B 0,C 180,E1 18381.913,E2 18381.913} C_VEL
LIN {X 0,Y 369.722,Z 384.67,A -85,B 0,C 180,E1 18377.794,E2 18377.794} C_VEL
LIN {X 0,Y 369.713,Z 384.668,A -85,B 0,C 180,E1 18373.768,E2 18373.768} C_VEL
LIN {X 0,Y 369.7,Z 384.664,A -85,B 0,C 180,E1 18369.811,E2 18369.811} C_VEL
LIN {X 0,Y 369.689,Z 384.661,A -85,B 0,C 180,E1 18365.899,E2 18365.899} C_VEL
LIN {X 0,Y 369.685,Z 384.662,A -85,B 0,C 180,E1 18361.86,E2 18361.86} C_VEL
LIN {X 0,Y 369.681,Z 384.667,A -85,B 0,C 180,E1 18357.83,E2 18357.83} C_VEL
LIN {X 0,Y 369.676,Z 384.671,A -85,B 0,C 180,E1 18353.79,E2 18353.79} C_VEL
LIN {X 0,Y 369.672,Z 384.673,A -85,B 0,C 180,E1 18349.717,E2 18349.717} C_VEL
LIN {X 0,Y 369.668,Z 384.673,A -85,B 0,C 180,E1 18345.592,E2 18345.592} C_VEL
LIN {X 0,Y 369.671,Z 384.672,A -85,B 0,C 180,E1 18341.552,E2 18341.552} C_VEL
LIN {X 0,Y 369.673,Z 384.638,A -85,B 0,C 180,E1 18337.582,E2 18337.582} C_VEL
LIN {X 0,Y 369.73,Z 384.946,A -85,B 0,C 180,E1 18335.729,E2 18335.729} C_VEL
LIN {X 0,Y 371.256,Z 388.479,A -85,B 0,C 180,E1 18334.646,E2 18334.646} C_VEL
LIN {X 0,Y 372.882,Z 390.476,A -85,B 0,C 180,E1 18333.912,E2 18333.912} C_VEL
LIN {X 0,Y 374.828,Z 394.257,A -85,B 0,C 180,E1 18332.862,E2 18332.862} C_VEL
LIN {X 0,Y 375.866,Z 395.521,A -85,B 0,C 180,E1 18332.428,E2 18332.428} C_VEL
LIN {X 0,Y 377.941,Z 399.443,A -85,B 0,C 180,E1 18331.391,E2 18331.391} C_VEL
LIN {X 0,Y 379.209,Z 401.623,A -85,B 0,C 180,E1 18330.805,E2 18330.805} C_VEL
LIN {X 0,Y 383.789,Z 409.646,A -85,B 0,C 180,E1 18328.773,E2 18328.773} C_VEL
LIN {X 0,Y 391.141,Z 423.831,A -85,B 0,C 180,E1 18325.649,E2 18325.649} C_VEL
LIN {X 0,Y 398.364,Z 438.723,A -85,B 0,C 180,E1 18322.78,E2 18322.78} C_VEL
LIN {X 0,Y 401.235,Z 443.768,A -85,B 0,C 180,E1 18322.079,E2 18322.079} C_VEL
LIN {X 0,Y 411.157,Z 460.26,A -85,B 0,C 180,E1 18320.105,E2 18320.105} C_VEL
LIN {X 0,Y 413.743,Z 465.164,A -85,B 0,C 180,E1 18319.602,E2 18319.602} C_VEL
LIN {X 0,Y 416.407,Z 496.05,A -85,B 0,C 180,E1 18318.446,E2 18318.446} C_VEL
LIN {X 0,Y 407.369,Z 720.295,A -85,B 0,C 180,E1 18314.095,E2 18314.095} C_VEL
LIN {X 0,Y 405.831,Z 749.731,A -85,B 0,C 180,E1 18313.449,E2 18313.449} C_VEL
LIN {X 0,Y 403.621,Z 771.98,A -85,B 0,C 180,E1 18312.754,E2 18312.754} C_VEL
LIN {X 0,Y 400.992,Z 792.125,A -85,B 0,C 180,E1 18311.901,E2 18311.901} C_VEL
LIN {X 0,Y 397.733,Z 813.577,A -85,B 0,C 180,E1 18310.725,E2 18310.725} C_VEL
LIN {X 0,Y 394.132,Z 834.809,A -85,B 0,C 180,E1 18309.264,E2 18309.264} C_VEL
LIN {X 0,Y 390.537,Z 854.329,A -85,B 0,C 180,E1 18307.63,E2 18307.63} C_VEL
LIN {X 0,Y 386.734,Z 873.78,A -85,B 0,C 180,E1 18305.659,E2 18305.659} C_VEL
LIN {X 0,Y 383.14,Z 891.796,A -85,B 0,C 180,E1 18303.497,E2 18303.497} C_VEL
LIN {X 0,Y 379.716,Z 909.048,A -85,B 0,C 180,E1 18301.068,E2 18301.068} C_VEL
LIN {X 0,Y 376.624,Z 925.346,A -85,B 0,C 180,E1 18298.37,E2 18298.37} C_VEL
LIN {X 0,Y 374.002,Z 940.04,A -85,B 0,C 180,E1 18295.492,E2 18295.492} C_VEL
LIN {X 0,Y 371.904,Z 953.282,A -85,B 0,C 180,E1 18292.441,E2 18292.441} C_VEL
LIN {X 0,Y 370.415,Z 964.509,A -85,B 0,C 180,E1 18289.39,E2 18289.39} C_VEL
LIN {X 0,Y 369.453,Z 973.807,A -85,B 0,C 180,E1 18286.346,E2 18286.346} C_VEL
LIN {X 0,Y 368.867,Z 981.74,A -85,B 0,C 180,E1 18283.16,E2 18283.16} C_VEL
LIN {X 0,Y 368.602,Z 987.871,A -85,B 0,C 180,E1 18280.05,E2 18280.05} C_VEL
LIN {X 0,Y 368.564,Z 992.157,A -85,B 0,C 180,E1 18277.012,E2 18277.012} C_VEL
LIN {X 0,Y 368.606,Z 994.984,A -85,B 0,C 180,E1 18274.044,E2 18274.044} C_VEL
LIN {X 0,Y 368.652,Z 996.198,A -85,B 0,C 180,E1 18271.088,E2 18271.088} C_VEL
LIN {X 0,Y 368.644,Z 996.087,A -85,B 0,C 180,E1 18268.291,E2 18268.291} C_VEL
LIN {X 0,Y 368.593,Z 994.335,A -85,B 0,C 180,E1 18265.177,E2 18265.177} C_VEL
LIN {X 0,Y 368.552,Z 991.411,A -85,B 0,C 180,E1 18262.362,E2 18262.362} C_VEL
LIN {X 0,Y 368.659,Z 986.524,A -85,B 0,C 180,E1 18259.216,E2 18259.216} C_VEL
LIN {X 0,Y 368.965,Z 979.994,A -85,B 0,C 180,E1 18256.046,E2 18256.046} C_VEL
LIN {X 0,Y 369.619,Z 971.977,A -85,B 0,C 180,E1 18253.016,E2 18253.016} C_VEL
LIN {X 0,Y 370.767,Z 961.67,A -85,B 0,C 180,E1 18249.794,E2 18249.794} C_VEL
LIN {X 0,Y 372.393,Z 950.086,A -85,B 0,C 180,E1 18246.757,E2 18246.757} C_VEL
LIN {X 0,Y 374.522,Z 936.952,A -85,B 0,C 180,E1 18243.868,E2 18243.868} C_VEL
LIN {X 0,Y 377.311,Z 921.596,A -85,B 0,C 180,E1 18240.983,E2 18240.983} C_VEL
LIN {X 0,Y 380.458,Z 905.304,A -85,B 0,C 180,E1 18238.373,E2 18238.373} C_VEL
LIN {X 0,Y 383.983,Z 887.61,A -85,B 0,C 180,E1 18235.96,E2 18235.96} C_VEL
LIN {X 0,Y 387.703,Z 868.791,A -85,B 0,C 180,E1 18233.807,E2 18233.807} C_VEL
LIN {X 0,Y 391.475,Z 849.188,A -85,B 0,C 180,E1 18231.922,E2 18231.922} C_VEL
LIN {X 0,Y 395.103,Z 829.207,A -85,B 0,C 180,E1 18230.32,E2 18230.32} C_VEL
LIN {X 0,Y 398.482,Z 808.977,A -85,B 0,C 180,E1 18228.999,E2 18228.999} C_VEL
LIN {X 0,Y 401.449,Z 788.618,A -85,B 0,C 180,E1 18227.94,E2 18227.94} C_VEL
LIN {X 0,Y 404.151,Z 767.017,A -85,B 0,C 180,E1 18227.074,E2 18227.074} C_VEL
LIN {X 0,Y 406.242,Z 744.194,A -85,B 0,C 180,E1 18226.407,E2 18226.407} C_VEL
LIN {X 0,Y 410.593,Z 637.372,A -85,B 0,C 180,E1 18224.293,E2 18224.293} C_VEL
LIN {X 0,Y 416.316,Z 493.623,A -85,B 0,C 180,E1 18221.494,E2 18221.494} C_VEL
LIN {X 0,Y 413.445,Z 464.384,A -85,B 0,C 180,E1 18220.354,E2 18220.354} C_VEL
LIN {X 0,Y 402.392,Z 445.551,A -85,B 0,C 180,E1 18218.176,E2 18218.176} C_VEL
LIN {X 0,Y 398.616,Z 439.331,A -85,B 0,C 180,E1 18217.34,E2 18217.34} C_VEL
LIN {X 0,Y 391.531,Z 424.654,A -85,B 0,C 180,E1 18214.536,E2 18214.536} C_VEL
LIN {X 0,Y 385.679,Z 413.38,A -85,B 0,C 180,E1 18212.103,E2 18212.103} C_VEL
LIN {X 0,Y 380.759,Z 404.319,A -85,B 0,C 180,E1 18209.929,E2 18209.929} C_VEL
LIN {X 0,Y 377.871,Z 399.359,A -85,B 0,C 180,E1 18208.615,E2 18208.615} C_VEL
LIN {X 0,Y 375.476,Z 394.946,A -85,B 0,C 180,E1 18207.431,E2 18207.431} C_VEL
LIN {X 0,Y 373.273,Z 391.624,A -85,B 0,C 180,E1 18206.401,E2 18206.401} C_VEL
LIN {X 0,Y 372.538,Z 389.842,A -85,B 0,C 180,E1 18205.943,E2 18205.943} C_VEL
LIN {X 0,Y 370.291,Z 386.867,A -85,B 0,C 180,E1 18204.884,E2 18204.884} C_VEL
LIN {X 0,Y 369.717,Z 384.876,A -85,B 0,C 180,E1 18204.271,E2 18204.271} C_VEL
LIN {X 0,Y 369.683,Z 384.681,A -85,B 0,C 180,E1 18201.082,E2 18201.082} C_VEL
LIN {X 0,Y 369.69,Z 384.687,A -85,B 0,C 180,E1 18197.145,E2 18197.145} C_VEL
LIN {X 0,Y 369.697,Z 384.685,A -85,B 0,C 180,E1 18193.131,E2 18193.131} C_VEL
LIN {X 0,Y 369.701,Z 384.683,A -85,B 0,C 180,E1 18189.024,E2 18189.024} C_VEL
LIN {X 0,Y 369.718,Z 384.682,A -85,B 0,C 180,E1 18185.12,E2 18185.12} C_VEL
LIN {X 0,Y 369.719,Z 384.68,A -85,B 0,C 180,E1 18180.929,E2 18180.929} C_VEL
LIN {X 0,Y 369.721,Z 384.671,A -85,B 0,C 180,E1 18176.893,E2 18176.893} C_VEL
LIN {X 0,Y 369.726,Z 384.664,A -85,B 0,C 180,E1 18172.697,E2 18172.697} C_VEL
LIN {X 0,Y 369.725,Z 384.661,A -85,B 0,C 180,E1 18168.614,E2 18168.614} C_VEL
LIN {X 0,Y 369.732,Z 384.661,A -85,B 0,C 180,E1 18164.471,E2 18164.471} C_VEL
LIN {X 0,Y 369.735,Z 384.66,A -85,B 0,C 180,E1 18160.407,E2 18160.407} C_VEL
LIN {X 0,Y 369.741,Z 384.66,A -85,B 0,C 180,E1 18156.407,E2 18156.407} C_VEL
LIN {X 0,Y 369.749,Z 384.663,A -85,B 0,C 180,E1 18152.148,E2 18152.148} C_VEL
LIN {X 0,Y 369.745,Z 384.67,A -85,B 0,C 180,E1 18148.105,E2 18148.105} C_VEL
LIN {X 0,Y 369.776,Z 384.959,A -85,B 0,C 180,E1 18145.824,E2 18145.824} C_VEL
LIN {X 0,Y 371.355,Z 388.616,A -85,B 0,C 180,E1 18144.628,E2 18144.628} C_VEL
LIN {X 0,Y 372.57,Z 390.253,A -85,B 0,C 180,E1 18144.004,E2 18144.004} C_VEL
LIN {X 0,Y 374.425,Z 393.924,A -85,B 0,C 180,E1 18142.878,E2 18142.878} C_VEL
LIN {X 0,Y 375.303,Z 395.432,A -85,B 0,C 180,E1 18142.404,E2 18142.404} C_VEL
LIN {X 0,Y 378.239,Z 401.072,A -85,B 0,C 180,E1 18140.818,E2 18140.818} C_VEL
LIN {X 0,Y 389.317,Z 415.32,A -85,B 0,C 180,E1 18138.205,E2 18138.205} C_VEL
LIN {X 0,Y 400.496,Z 431.037,A -85,B 0,C 180,E1 18135.825,E2 18135.825} C_VEL
LIN {X 0,Y 411.863,Z 448.471,A -85,B 0,C 180,E1 18133.61,E2 18133.61} C_VEL
LIN {X 0,Y 414.643,Z 453.301,A -85,B 0,C 180,E1 18133.088,E2 18133.088} C_VEL
LIN {X 0,Y 407.563,Z 663.77,A -85,B 0,C 180,E1 18129.279,E2 18129.279} C_VEL
LIN {X 0,Y 406.391,Z 683.961,A -85,B 0,C 180,E1 18128.666,E2 18128.666} C_VEL
LIN {X 0,Y 404.541,Z 704.268,A -85,B 0,C 180,E1 18127.798,E2 18127.798} C_VEL
LIN {X 0,Y 402.15,Z 723.532,A -85,B 0,C 180,E1 18126.718,E2 18126.718} C_VEL
LIN {X 0,Y 399.319,Z 741.904,A -85,B 0,C 180,E1 18125.422,E2 18125.422} C_VEL
LIN {X 0,Y 396.086,Z 759.245,A -85,B 0,C 180,E1 18123.905,E2 18123.905} C_VEL
LIN {X 0,Y 392.6,Z 775.772,A -85,B 0,C 180,E1 18122.155,E2 18122.155} C_VEL
LIN {X 0,Y 388.835,Z 791.939,A -85,B 0,C 180,E1 18120.091,E2 18120.091} C_VEL
LIN {X 0,Y 385.415,Z 805.635,A -85,B 0,C 180,E1 18118.002,E2 18118.002} C_VEL
LIN {X 0,Y 381.956,Z 818.835,A -85,B 0,C 180,E1 18115.586,E2 18115.586} C_VEL
LIN {X 0,Y 378.766,Z 830.587,A -85,B 0,C 180,E1 18112.994,E2 18112.994} C_VEL
LIN {X 0,Y 375.927,Z 841.265,A -85,B 0,C 180,E1 18110.135,E2 18110.135} C_VEL
LIN {X 0,Y 373.477,Z 850.818,A -85,B 0,C 180,E1 18106.964,E2 18106.964} C_VEL
LIN {X 0,Y 373.444,Z 850.955,A -85,B 0,C 180,E1 18106.913,E2 18106.913} C_VEL
LIN {X 0,Y 371.817,Z 854.003,A -85,B 0,C 180,E1 18105.84,E2 18105.84} C_VEL
LIN {X 0,Y 364.265,Z 861.697,A -85,B 0,C 180,E1 18102.986,E2 18102.986} C_VEL
LIN {X 0,Y 363.135,Z 863.566,A -85,B 0,C 180,E1 18101.997,E2 18101.997} C_VEL
LIN {X 0,Y 362.181,Z 868.44,A -85,B 0,C 180,E1 18098.572,E2 18098.572} C_VEL
LIN {X 0,Y 361.647,Z 871.583,A -85,B 0,C 180,E1 18095.234,E2 18095.234} C_VEL
LIN {X 0,Y 361.418,Z 873.209,A -85,B 0,C 180,E1 18091.902,E2 18091.902} C_VEL
LIN {X 0,Y 361.39,Z 873.296,A -85,B 0,C 180,E1 18088.573,E2 18088.573} C_VEL
LIN {X 0,Y 361.584,Z 871.942,A -85,B 0,C 180,E1 18085.241,E2 18085.241} C_VEL
LIN {X 0,Y 362.096,Z 868.917,A -85,B 0,C 180,E1 18081.745,E2 18081.745} C_VEL
LIN {X 0,Y 362.973,Z 864.402,A -85,B 0,C 180,E1 18078.4,E2 18078.4} C_VEL
LIN {X 0,Y 364.355,Z 858.497,A -85,B 0,C 180,E1 18075.215,E2 18075.215} C_VEL
LIN {X 0,Y 366.296,Z 850.773,A -85,B 0,C 180,E1 18072.035,E2 18072.035} C_VEL
LIN {X 0,Y 368.799,Z 841.61,A -85,B 0,C 180,E1 18069.032,E2 18069.032} C_VEL
LIN {X 0,Y 371.757,Z 831.065,A -85,B 0,C 180,E1 18066.209,E2 18066.209} C_VEL
LIN {X 0,Y 375.158,Z 819.127,A -85,B 0,C 180,E1 18063.573,E2 18063.573} C_VEL
LIN {X 0,Y 378.844,Z 805.794,A -85,B 0,C 180,E1 18061.122,E2 18061.122} C_VEL
LIN {X 0,Y 382.734,Z 790.849,A -85,B 0,C 180,E1 18058.854,E2 18058.854} C_VEL
LIN {X 0,Y 386.423,Z 775.45,A -85,B 0,C 180,E1 18056.913,E2 18056.913} C_VEL
LIN {X 0,Y 390.204,Z 757.94,A -85,B 0,C 180,E1 18055.082,E2 18055.082} C_VEL
LIN {X 0,Y 393.62,Z 739.814,A -85,B 0,C 180,E1 18053.534,E2 18053.534} C_VEL
LIN {X 0,Y 396.449,Z 722.058,A -85,B 0,C 180,E1 18052.299,E2 18052.299} C_VEL
LIN {X 0,Y 398.773,Z 703.281,A -85,B 0,C 180,E1 18051.27,E2 18051.27} C_VEL
LIN {X 0,Y 400.598,Z 683.199,A -85,B 0,C 180,E1 18050.43,E2 18050.43} C_VEL
LIN {X 0,Y 401.808,Z 661.607,A -85,B 0,C 180,E1 18049.802,E2 18049.802} C_VEL
LIN {X 0,Y 409.008,Z 456.468,A -85,B 0,C 180,E1 18046.049,E2 18046.049} C_VEL
LIN {X 0,Y 397.256,Z 437.956,A -85,B 0,C 180,E1 18043.701,E2 18043.701} C_VEL
LIN {X 0,Y 385.318,Z 421.01,A -85,B 0,C 180,E1 18041.084,E2 18041.084} C_VEL
LIN {X 0,Y 373.506,Z 405.722,A -85,B 0,C 180,E1 18038.198,E2 18038.198} C_VEL
LIN {X 0,Y 370.155,Z 401.381,A -85,B 0,C 180,E1 18037.234,E2 18037.234} C_VEL
LIN {X 0,Y 366.87,Z 395.356,A -85,B 0,C 180,E1 18035.295,E2 18035.295} C_VEL
LIN {X 0,Y 365.008,Z 392.165,A -85,B 0,C 180,E1 18034.164,E2 18034.164} C_VEL
LIN {X 0,Y 364.352,Z 390.576,A -85,B 0,C 180,E1 18033.665,E2 18033.665} C_VEL
LIN {X 0,Y 362.203,Z 387.407,A -85,B 0,C 180,E1 18032.381,E2 18032.381} C_VEL
LIN {X 0,Y 361.816,Z 385.73,A -85,B 0,C 180,E1 18031.719,E2 18031.719} C_VEL
LIN {X 0,Y 361.809,Z 385.65,A -85,B 0,C 180,E1 18027.663,E2 18027.663} C_VEL
LIN {X 0,Y 361.803,Z 385.646,A -85,B 0,C 180,E1 18023.449,E2 18023.449} C_VEL
LIN {X 0,Y 361.799,Z 385.645,A -85,B 0,C 180,E1 18019.368,E2 18019.368} C_VEL
LIN {X 0,Y 361.801,Z 385.646,A -85,B 0,C 180,E1 18015.221,E2 18015.221} C_VEL
LIN {X 0,Y 361.791,Z 385.649,A -85,B 0,C 180,E1 18011.155,E2 18011.155} C_VEL
LIN {X 0,Y 361.795,Z 385.65,A -85,B 0,C 180,E1 18006.985,E2 18006.985} C_VEL
LIN {X 0,Y 361.781,Z 385.656,A -85,B 0,C 180,E1 18002.852,E2 18002.852} C_VEL
LIN {X 0,Y 361.783,Z 385.663,A -85,B 0,C 180,E1 17998.733,E2 17998.733} C_VEL
LIN {X 0,Y 361.778,Z 385.668,A -85,B 0,C 180,E1 17994.609,E2 17994.609} C_VEL
LIN {X 0,Y 361.779,Z 385.67,A -85,B 0,C 180,E1 17990.596,E2 17990.596} C_VEL
LIN {X 0,Y 361.776,Z 385.669,A -85,B 0,C 180,E1 17986.414,E2 17986.414} C_VEL
LIN {X 0,Y 361.769,Z 385.664,A -85,B 0,C 180,E1 17982.301,E2 17982.301} C_VEL
LIN {X 0,Y 361.775,Z 385.718,A -85,B 0,C 180,E1 17978.072,E2 17978.072} C_VEL
LIN {X 0,Y 361.973,Z 386.809,A -85,B 0,C 180,E1 17977.593,E2 17977.593} C_VEL
LIN {X 0,Y 363.746,Z 389.964,A -85,B 0,C 180,E1 17976.511,E2 17976.511} C_VEL
LIN {X 0,Y 365.009,Z 391.364,A -85,B 0,C 180,E1 17975.912,E2 17975.912} C_VEL
LIN {X 0,Y 366.858,Z 395.099,A -85,B 0,C 180,E1 17974.793,E2 17974.793} C_VEL
LIN {X 0,Y 368.07,Z 396.559,A -85,B 0,C 180,E1 17974.238,E2 17974.238} C_VEL
LIN {X 0,Y 370.316,Z 400.777,A -85,B 0,C 180,E1 17973.025,E2 17973.025} C_VEL
LIN {X 0,Y 371.506,Z 402.883,A -85,B 0,C 180,E1 17972.425,E2 17972.425} C_VEL
LIN {X 0,Y 374.305,Z 407.687,A -85,B 0,C 180,E1 17971.087,E2 17971.087} C_VEL
LIN {X 0,Y 379.099,Z 416.425,A -85,B 0,C 180,E1 17968.873,E2 17968.873} C_VEL
LIN {X 0,Y 385.505,Z 428.772,A -85,B 0,C 180,E1 17966.087,E2 17966.087} C_VEL
LIN {X 0,Y 390.957,Z 439.702,A -85,B 0,C 180,E1 17963.947,E2 17963.947} C_VEL
LIN {X 0,Y 402.747,Z 458.779,A -85,B 0,C 180,E1 17961.433,E2 17961.433} C_VEL
LIN {X 0,Y 408.42,Z 469.126,A -85,B 0,C 180,E1 17960.286,E2 17960.286} C_VEL
LIN {X 0,Y 410.734,Z 497.313,A -85,B 0,C 180,E1 17959.214,E2 17959.214} C_VEL
LIN {X 0,Y 401.291,Z 721.629,A -85,B 0,C 180,E1 17954.817,E2 17954.817} C_VEL
LIN {X 0,Y 399.761,Z 748.988,A -85,B 0,C 180,E1 17954.204,E2 17954.204} C_VEL
LIN {X 0,Y 397.448,Z 771.343,A -85,B 0,C 180,E1 17953.495,E2 17953.495} C_VEL
LIN {X 0,Y 394.75,Z 791.19,A -85,B 0,C 180,E1 17952.648,E2 17952.648} C_VEL
LIN {X 0,Y 391.475,Z 811.859,A -85,B 0,C 180,E1 17951.508,E2 17951.508} C_VEL
LIN {X 0,Y 387.883,Z 832.138,A -85,B 0,C 180,E1 17950.119,E2 17950.119} C_VEL
LIN {X 0,Y 383.912,Z 852.784,A -85,B 0,C 180,E1 17948.379,E2 17948.379} C_VEL
LIN {X 0,Y 380.06,Z 871.435,A -85,B 0,C 180,E1 17946.478,E2 17946.478} C_VEL
LIN {X 0,Y 376.175,Z 889.915,A -85,B 0,C 180,E1 17944.247,E2 17944.247} C_VEL
LIN {X 0,Y 372.603,Z 906.993,A -85,B 0,C 180,E1 17941.82,E2 17941.82} C_VEL
LIN {X 0,Y 369.381,Z 922.884,A -85,B 0,C 180,E1 17939.156,E2 17939.156} C_VEL
LIN {X 0,Y 366.542,Z 937.755,A -85,B 0,C 180,E1 17936.223,E2 17936.223} C_VEL
LIN {X 0,Y 364.271,Z 951.159,A -85,B 0,C 180,E1 17933.109,E2 17933.109} C_VEL
LIN {X 0,Y 362.652,Z 962.535,A -85,B 0,C 180,E1 17929.99,E2 17929.99} C_VEL
LIN {X 0,Y 361.601,Z 971.913,A -85,B 0,C 180,E1 17926.877,E2 17926.877} C_VEL
LIN {X 0,Y 360.941,Z 980.334,A -85,B 0,C 180,E1 17923.455,E2 17923.455} C_VEL
LIN {X 0,Y 360.677,Z 986.583,A -85,B 0,C 180,E1 17920.219,E2 17920.219} C_VEL
LIN {X 0,Y 360.64,Z 990.799,A -85,B 0,C 180,E1 17917.167,E2 17917.167} C_VEL
LIN {X 0,Y 360.705,Z 993.645,A -85,B 0,C 180,E1 17914.133,E2 17914.133} C_VEL
LIN {X 0,Y 360.763,Z 994.869,A -85,B 0,C 180,E1 17911.112,E2 17911.112} C_VEL
LIN {X 0,Y 360.752,Z 994.757,A -85,B 0,C 180,E1 17908.254,E2 17908.254} C_VEL
LIN {X 0,Y 360.69,Z 993.124,A -85,B 0,C 180,E1 17905.231,E2 17905.231} C_VEL
LIN {X 0,Y 360.635,Z 990.239,A -85,B 0,C 180,E1 17902.354,E2 17902.354} C_VEL
LIN {X 0,Y 360.724,Z 985.136,A -85,B 0,C 180,E1 17898.976,E2 17898.976} C_VEL
LIN {X 0,Y 361.033,Z 978.576,A -85,B 0,C 180,E1 17895.733,E2 17895.733} C_VEL
LIN {X 0,Y 361.723,Z 970.534,A -85,B 0,C 180,E1 17892.633,E2 17892.633} C_VEL
LIN {X 0,Y 363.026,Z 959.68,A -85,B 0,C 180,E1 17889.191,E2 17889.191} C_VEL
LIN {X 0,Y 364.8,Z 947.893,A -85,B 0,C 180,E1 17886.072,E2 17886.072} C_VEL
LIN {X 0,Y 367.102,Z 934.661,A -85,B 0,C 180,E1 17883.123,E2 17883.123} C_VEL
LIN {X 0,Y 369.911,Z 920.11,A -85,B 0,C 180,E1 17880.358,E2 17880.358} C_VEL
LIN {X 0,Y 373.274,Z 903.794,A -85,B 0,C 180,E1 17877.702,E2 17877.702} C_VEL
LIN {X 0,Y 377.013,Z 886.01,A -85,B 0,C 180,E1 17875.241,E2 17875.241} C_VEL
LIN {X 0,Y 380.94,Z 867.153,A -85,B 0,C 180,E1 17873.059,E2 17873.059} C_VEL
LIN {X 0,Y 384.895,Z 847.568,A -85,B 0,C 180,E1 17871.16,E2 17871.16} C_VEL
LIN {X 0,Y 388.798,Z 827.074,A -85,B 0,C 180,E1 17869.513,E2 17869.513} C_VEL
LIN {X 0,Y 392.472,Z 805.919,A -85,B 0,C 180,E1 17868.134,E2 17868.134} C_VEL
LIN {X 0,Y 395.691,Z 784.311,A -85,B 0,C 180,E1 17867.035,E2 17867.035} C_VEL
LIN {X 0,Y 398.461,Z 762.166,A -85,B 0,C 180,E1 17866.191,E2 17866.191} C_VEL
LIN {X 0,Y 400.431,Z 739.116,A -85,B 0,C 180,E1 17865.554,E2 17865.554} C_VEL
LIN {X 0,Y 409.033,Z 535.822,A -85,B 0,C 180,E1 17861.54,E2 17861.54} C_VEL
LIN {X 0,Y 410.624,Z 494.717,A -85,B 0,C 180,E1 17860.718,E2 17860.718} C_VEL
LIN {X 0,Y 408.151,Z 468.439,A -85,B 0,C 180,E1 17859.677,E2 17859.677} C_VEL
LIN {X 0,Y 398.115,Z 451.177,A -85,B 0,C 180,E1 17857.633,E2 17857.633} C_VEL
LIN {X 0,Y 390.316,Z 438.723,A -85,B 0,C 180,E1 17855.917,E2 17855.917} C_VEL
LIN {X 0,Y 383.064,Z 423.869,A -85,B 0,C 180,E1 17852.882,E2 17852.882} C_VEL
LIN {X 0,Y 376.178,Z 410.858,A -85,B 0,C 180,E1 17849.804,E2 17849.804} C_VEL
LIN {X 0,Y 372.64,Z 404.951,A -85,B 0,C 180,E1 17848.179,E2 17848.179} C_VEL
LIN {X 0,Y 370.342,Z 400.797,A -85,B 0,C 180,E1 17847.021,E2 17847.021} C_VEL
LIN {X 0,Y 368.234,Z 397.055,A -85,B 0,C 180,E1 17845.922,E2 17845.922} C_VEL
LIN {X 0,Y 365.354,Z 392.434,A -85,B 0,C 180,E1 17844.408,E2 17844.408} C_VEL
LIN {X 0,Y 364.635,Z 390.843,A -85,B 0,C 180,E1 17843.943,E2 17843.943} C_VEL
LIN {X 0,Y 362.302,Z 387.745,A -85,B 0,C 180,E1 17842.728,E2 17842.728} C_VEL
LIN {X 0,Y 361.784,Z 385.852,A -85,B 0,C 180,E1 17842.077,E2 17842.077} C_VEL
LIN {X 0,Y 361.749,Z 385.661,A -85,B 0,C 180,E1 17838.032,E2 17838.032} C_VEL
LIN {X 0,Y 361.739,Z 385.664,A -85,B 0,C 180,E1 17834.054,E2 17834.054} C_VEL
LIN {X 0,Y 361.74,Z 385.663,A -85,B 0,C 180,E1 17830.028,E2 17830.028} C_VEL
LIN {X 0,Y 361.738,Z 385.661,A -85,B 0,C 180,E1 17826.029,E2 17826.029} C_VEL
LIN {X 0,Y 361.742,Z 385.657,A -85,B 0,C 180,E1 17821.9,E2 17821.9} C_VEL
LIN {X 0,Y 361.744,Z 385.652,A -85,B 0,C 180,E1 17817.782,E2 17817.782} C_VEL
LIN {X 0,Y 361.746,Z 385.648,A -85,B 0,C 180,E1 17813.652,E2 17813.652} C_VEL
LIN {X 0,Y 361.75,Z 385.648,A -85,B 0,C 180,E1 17809.65,E2 17809.65} C_VEL
LIN {X 0,Y 361.751,Z 385.652,A -85,B 0,C 180,E1 17805.596,E2 17805.596} C_VEL
LIN {X 0,Y 361.757,Z 385.654,A -85,B 0,C 180,E1 17801.425,E2 17801.425} C_VEL
LIN {X 0,Y 361.76,Z 385.654,A -85,B 0,C 180,E1 17797.373,E2 17797.373} C_VEL
LIN {X 0,Y 361.764,Z 385.653,A -85,B 0,C 180,E1 17793.205,E2 17793.205} C_VEL
LIN {X 0,Y 361.767,Z 385.654,A -85,B 0,C 180,E1 17789.064,E2 17789.064} C_VEL
LIN {X 0,Y 361.843,Z 385.957,A -85,B 0,C 180,E1 17787.958,E2 17787.958} C_VEL
LIN {X 0,Y 363.203,Z 389.321,A -85,B 0,C 180,E1 17786.782,E2 17786.782} C_VEL
LIN {X 0,Y 364.69,Z 391.118,A -85,B 0,C 180,E1 17785.992,E2 17785.992} C_VEL
LIN {X 0,Y 366.336,Z 394.713,A -85,B 0,C 180,E1 17784.837,E2 17784.837} C_VEL
LIN {X 0,Y 367.503,Z 396.451,A -85,B 0,C 180,E1 17784.2,E2 17784.2} C_VEL
LIN {X 0,Y 369.737,Z 400.442,A -85,B 0,C 180,E1 17782.907,E2 17782.907} C_VEL
LIN {X 0,Y 371.123,Z 403.016,A -85,B 0,C 180,E1 17782.296,E2 17782.296} C_VEL
LIN {X 0,Y 376.141,Z 409.23,A -85,B 0,C 180,E1 17780.999,E2 17780.999} C_VEL
LIN {X 0,Y 386.072,Z 422.134,A -85,B 0,C 180,E1 17778.619,E2 17778.619} C_VEL
LIN {X 0,Y 397.502,Z 438.388,A -85,B 0,C 180,E1 17776.133,E2 17776.133} C_VEL
LIN {X 0,Y 409.012,Z 456.527,A -85,B 0,C 180,E1 17773.844,E2 17773.844} C_VEL
LIN {X 0,Y 401.654,Z 664.657,A -85,B 0,C 180,E1 17770.033,E2 17770.033} C_VEL
LIN {X 0,Y 400.437,Z 684.839,A -85,B 0,C 180,E1 17769.414,E2 17769.414} C_VEL
LIN {X 0,Y 398.563,Z 704.747,A -85,B 0,C 180,E1 17768.56,E2 17768.56} C_VEL
LIN {X 0,Y 396.254,Z 723.064,A -85,B 0,C 180,E1 17767.539,E2 17767.539} C_VEL
LIN {X 0,Y 393.279,Z 741.649,A -85,B 0,C 180,E1 17766.23,E2 17766.23} C_VEL
LIN {X 0,Y 389.905,Z 759.257,A -85,B 0,C 180,E1 17764.696,E2 17764.696} C_VEL
LIN {X 0,Y 386.26,Z 776.002,A -85,B 0,C 180,E1 17762.925,E2 17762.925} C_VEL
LIN {X 0,Y 382.444,Z 791.822,A -85,B 0,C 180,E1 17760.908,E2 17760.908} C_VEL
LIN {X 0,Y 378.712,Z 806.185,A -85,B 0,C 180,E1 17758.715,E2 17758.715} C_VEL
LIN {X 0,Y 374.838,Z 820.248,A -85,B 0,C 180,E1 17756.109,E2 17756.109} C_VEL
LIN {X 0,Y 371.486,Z 831.979,A -85,B 0,C 180,E1 17753.472,E2 17753.472} C_VEL
LIN {X 0,Y 368.538,Z 842.474,A -85,B 0,C 180,E1 17750.609,E2 17750.609} C_VEL
LIN {X 0,Y 366.005,Z 851.767,A -85,B 0,C 180,E1 17747.485,E2 17747.485} C_VEL
LIN {X 0,Y 364.136,Z 859.258,A -85,B 0,C 180,E1 17744.305,E2 17744.305} C_VEL
LIN {X 0,Y 363.135,Z 863.566,A -85,B 0,C 180,E1 17741.997,E2 17741.997} C_VEL
LIN {X 0,Y 361.769,Z 865.669,A -85,B 0,C 180,E1 17740.833,E2 17740.833} C_VEL
LIN {X 0,Y 354.885,Z 870.799,A -85,B 0,C 180,E1 17737.72,E2 17737.72} C_VEL
LIN {X 0,Y 353.958,Z 871.872,A -85,B 0,C 180,E1 17736.665,E2 17736.665} C_VEL
LIN {X 0,Y 353.576,Z 874.122,A -85,B 0,C 180,E1 17733.079,E2 17733.079} C_VEL
LIN {X 0,Y 353.492,Z 874.762,A -85,B 0,C 180,E1 17729.675,E2 17729.675} C_VEL
LIN {X 0,Y 353.62,Z 873.927,A -85,B 0,C 180,E1 17726.271,E2 17726.271} C_VEL
LIN {X 0,Y 354.031,Z 871.556,A -85,B 0,C 180,E1 17722.862,E2 17722.862} C_VEL
LIN {X 0,Y 354.783,Z 867.647,A -85,B 0,C 180,E1 17719.445,E2 17719.445} C_VEL
LIN {X 0,Y 356.089,Z 862.061,A -85,B 0,C 180,E1 17716.027,E2 17716.027} C_VEL
LIN {X 0,Y 357.947,Z 855.034,A -85,B 0,C 180,E1 17712.778,E2 17712.778} C_VEL
LIN {X 0,Y 360.501,Z 846.122,A -85,B 0,C 180,E1 17709.547,E2 17709.547} C_VEL
LIN {X 0,Y 363.602,Z 835.625,A -85,B 0,C 180,E1 17706.503,E2 17706.503} C_VEL
LIN {X 0,Y 366.982,Z 824.251,A -85,B 0,C 180,E1 17703.81,E2 17703.81} C_VEL
LIN {X 0,Y 370.854,Z 810.921,A -85,B 0,C 180,E1 17701.192,E2 17701.192} C_VEL
LIN {X 0,Y 375.036,Z 795.896,A -85,B 0,C 180,E1 17698.758,E2 17698.758} C_VEL
LIN {X 0,Y 379.034,Z 780.367,A -85,B 0,C 180,E1 17696.672,E2 17696.672} C_VEL
LIN {X 0,Y 382.953,Z 763.603,A -85,B 0,C 180,E1 17694.808,E2 17694.808} C_VEL
LIN {X 0,Y 386.506,Z 746.07,A -85,B 0,C 180,E1 17693.215,E2 17693.215} C_VEL
LIN {X 0,Y 389.565,Z 728.187,A -85,B 0,C 180,E1 17691.887,E2 17691.887} C_VEL
LIN {X 0,Y 392.346,Z 708.233,A -85,B 0,C 180,E1 17690.712,E2 17690.712} C_VEL
LIN {X 0,Y 394.371,Z 688.825,A -85,B 0,C 180,E1 17689.832,E2 17689.832} C_VEL
LIN {X 0,Y 395.766,Z 668.191,A -85,B 0,C 180,E1 17689.159,E2 17689.159} C_VEL
LIN {X 0,Y 397.113,Z 629.706,A -85,B 0,C 180,E1 17688.394,E2 17688.394} C_VEL
